KUKA KRL program: f1_Kuka_APT228T02S28.SRC

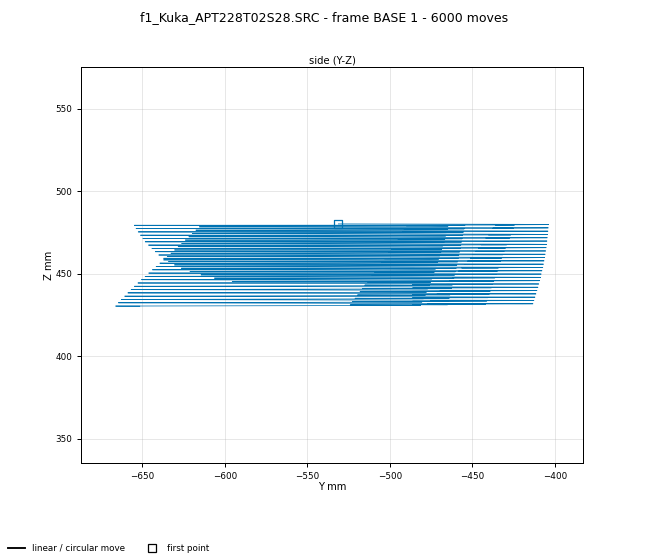
[picture p0: tool path of f1_Kuka_APT228T02S28.SRC in frame BASE 1, 6000 of 6001 moves have a stored position in this frame; points joined in program order, loops and branches not executed]
&ACCESS RVP
&REL 2
&PARAM TEMPLATE = C:\KRC\Roboter\Template\vorgabe
&PARAM EDITMASK = *
DEF f1_Kuka_APT228T02S28()


;FOLD INI;%{PE}%V3.2.0,%MKUKATPBASIS,%CINIT,%VCOMMON,%P
  ;FOLD BAS INI;%{E}%V3.2.0,%MKUKATPBASIS,%CINIT,%VINIT,%P
    GLOBAL INTERRUPT DECL 3 WHEN $STOPMESS==TRUE DO IR_STOPM ( )
    INTERRUPT ON 3
    BAS (#INITMOV,0 )
  ;ENDFOLD (BAS INI)
  ;FOLD USER INI;%{E}%V3.2.0,%MKUKATPUSER,%CINIT,%VINIT,%P
    ;Make your modifications here
  ;ENDFOLD (USER INI)
;ENDFOLD (INI)


;*** Make Null PTP Move
  PTP $pos_act

;*** Auto Load The Correct TOOL Data
  $tool=tool_data[2]

;*** Auto Load The Correct BASE Data
  $base=base_data[1]

  $ADVANCE = 5

;*** Restate Last Velocity
MMPM(30000.0)
SetRPM(8000)
LIN {X 0.012,Y -531.223,Z 480.140,A 0.000,B 0.000,C 90.000,E1 241.129} C_DIS
LIN {X -0.132,Y -524.473,Z 480.128,A 0.000,B 0.000,C 90.000,E1 239.125} C_DIS
LIN {X -0.042,Y -519.669,Z 480.120,A 0.000,B 0.000,C 90.000,E1 237.661} C_DIS
LIN {X -0.136,Y -515.820,Z 480.114,A 0.000,B 0.000,C 90.000,E1 236.501} C_DIS
LIN {X 0.003,Y -511.801,Z 480.107,A 0.000,B 0.000,C 90.000,E1 235.308} C_DIS
LIN {X 0.099,Y -503.620,Z 480.094,A 0.000,B 0.000,C 90.000,E1 232.924} C_DIS
LIN {X 0.015,Y -495.240,Z 480.079,A 0.000,B 0.000,C 90.000,E1 230.231} C_DIS
LIN {X 0.077,Y -489.925,Z 480.069,A 0.000,B 0.000,C 90.000,E1 228.405} C_DIS
LIN {X -0.155,Y -485.610,Z 480.061,A 0.000,B 0.000,C 90.000,E1 226.905} C_DIS
LIN {X 0.222,Y -481.353,Z 480.052,A 0.000,B 0.000,C 90.000,E1 225.324} C_DIS
LIN {X 0.174,Y -474.838,Z 480.038,A 0.000,B 0.000,C 90.000,E1 222.852} C_DIS
LIN {X -0.124,Y -469.500,Z 480.026,A 0.000,B 0.000,C 90.000,E1 220.701} C_DIS
LIN {X -0.093,Y -463.775,Z 480.012,A 0.000,B 0.000,C 90.000,E1 218.177} C_DIS
LIN {X 0.094,Y -459.135,Z 480.000,A 0.000,B 0.000,C 90.000,E1 215.931} C_DIS
LIN {X -0.017,Y -454.671,Z 479.987,A 0.000,B 0.000,C 90.000,E1 213.706} C_DIS
LIN {X -0.201,Y -450.942,Z 479.977,A 0.000,B 0.000,C 90.000,E1 211.799} C_DIS
LIN {X 0.216,Y -447.979,Z 479.968,A 0.000,B 0.000,C 90.000,E1 210.129} C_DIS
LIN {X -0.195,Y -444.403,Z 479.957,A 0.000,B 0.000,C 90.000,E1 208.231} C_DIS
LIN {X 0.099,Y -440.825,Z 479.946,A 0.000,B 0.000,C 90.000,E1 206.232} C_DIS
LIN {X 0.104,Y -437.235,Z 479.935,A 0.000,B 0.000,C 90.000,E1 204.259} C_DIS
LIN {X 0.071,Y -433.639,Z 479.924,A 0.000,B 0.000,C 90.000,E1 202.280} C_DIS
LIN {X -0.019,Y -428.986,Z 479.909,A 0.000,B 0.000,C 90.000,E1 199.631} C_DIS
LIN {X 0.061,Y -425.308,Z 479.896,A 0.000,B 0.000,C 90.000,E1 197.275} C_DIS
LIN {X 0.036,Y -421.007,Z 479.879,A 0.000,B 0.000,C 90.000,E1 194.245} C_DIS
LIN {X -0.197,Y -418.417,Z 479.868,A 0.000,B 0.000,C 90.000,E1 192.243} C_DIS
LIN {X -0.066,Y -415.176,Z 479.853,A 0.000,B 0.000,C 90.000,E1 189.500} C_DIS
LIN {X -0.177,Y -412.255,Z 479.838,A 0.000,B 0.000,C 90.000,E1 186.777} C_DIS
LIN {X -0.098,Y -409.929,Z 479.824,A 0.000,B 0.000,C 90.000,E1 184.359} C_DIS
LIN {X -0.138,Y -407.863,Z 479.811,A 0.000,B 0.000,C 90.000,E1 181.949} C_DIS
LIN {X 0.112,Y -405.824,Z 479.793,A 0.000,B 0.000,C 90.000,E1 178.797} C_DIS
LIN {X -0.117,Y -404.326,Z 479.774,A 0.000,B 0.000,C 90.000,E1 175.355} C_DIS
LIN {X 0.145,Y -403.885,Z 479.755,A 0.000,B 0.000,C 90.000,E1 171.837} C_DIS
LIN {X -0.149,Y -404.385,Z 479.735,A 0.000,B 0.000,C 90.000,E1 168.398} C_DIS
LIN {X 0.042,Y -405.380,Z 479.720,A 0.000,B 0.000,C 90.000,E1 165.589} C_DIS
LIN {X -0.122,Y -407.093,Z 479.703,A 0.000,B 0.000,C 90.000,E1 162.489} C_DIS
LIN {X -0.085,Y -408.847,Z 479.689,A 0.000,B 0.000,C 90.000,E1 160.061} C_DIS
LIN {X 0.144,Y -410.958,Z 479.676,A 0.000,B 0.000,C 90.000,E1 157.614} C_DIS
LIN {X 0.241,Y -413.011,Z 479.664,A 0.000,B 0.000,C 90.000,E1 155.537} C_DIS
LIN {X 0.018,Y -415.202,Z 479.653,A 0.000,B 0.000,C 90.000,E1 153.512} C_DIS
LIN {X -0.097,Y -417.093,Z 479.643,A 0.000,B 0.000,C 90.000,E1 151.820} C_DIS
LIN {X 0.146,Y -419.334,Z 479.632,A 0.000,B 0.000,C 90.000,E1 149.744} C_DIS
LIN {X -0.085,Y -421.583,Z 479.621,A 0.000,B 0.000,C 90.000,E1 147.740} C_DIS
LIN {X 0.013,Y -423.053,Z 479.613,A 0.000,B 0.000,C 90.000,E1 146.373} C_DIS
LIN {X 0.000,Y -424.931,Z 479.604,A 0.000,B 0.000,C 90.000,E1 144.689} C_DIS
LIN {X -0.113,Y -427.584,Z 479.591,A 0.000,B 0.000,C 90.000,E1 142.351} C_DIS
LIN {X 0.145,Y -429.546,Z 479.582,A 0.000,B 0.000,C 90.000,E1 140.642} C_DIS
LIN {X 0.089,Y -431.818,Z 479.570,A 0.000,B 0.000,C 90.000,E1 138.647} C_DIS
LIN {X 0.135,Y -433.268,Z 479.563,A 0.000,B 0.000,C 90.000,E1 137.310} C_DIS
LIN {X 0.207,Y -434.411,Z 479.556,A 0.000,B 0.000,C 90.000,E1 135.972} C_DIS
LIN {X 0.040,Y -435.117,Z 479.550,A 0.000,B 0.000,C 90.000,E1 135.000} C_DIS
LIN {X -0.120,Y -435.679,Z 479.545,A 0.000,B 0.000,C 90.000,E1 134.028} C_DIS
LIN {X 0.040,Y -436.073,Z 479.539,A 0.000,B 0.000,C 90.000,E1 133.014} C_DIS
LIN {X 0.208,Y -436.280,Z 479.534,A 0.000,B 0.000,C 90.000,E1 132.000} C_DIS
LIN {X -0.241,Y -436.121,Z 479.528,A 0.000,B 0.000,C 90.000,E1 131.067} C_DIS
LIN {X 0.250,Y -435.587,Z 479.523,A 0.000,B 0.000,C 90.000,E1 130.011} C_DIS
LIN {X -0.224,Y -434.407,Z 479.515,A 0.000,B 0.000,C 90.000,E1 128.749} C_DIS
LIN {X 0.045,Y -433.713,Z 479.511,A 0.000,B 0.000,C 90.000,E1 128.051} C_DIS
LIN {X 0.146,Y -431.523,Z 479.502,A 0.000,B 0.000,C 90.000,E1 126.377} C_DIS
LIN {X 0.291,Y -429.397,Z 479.495,A 0.000,B 0.000,C 90.000,E1 125.025} C_DIS
LIN {X 0.154,Y -427.076,Z 479.487,A 0.000,B 0.000,C 90.000,E1 123.706} C_DIS
LIN {X 0.257,Y -424.569,Z 479.480,A 0.000,B 0.000,C 90.000,E1 122.339} C_DIS
LIN {X 0.218,Y -424.582,Z 479.480,A 0.000,B 0.000,C 90.000,E1 122.339} C_DIS
LIN {X -0.108,Y -430.513,Z 479.469,A 0.000,B 0.000,C 90.000,E1 120.384} C_DIS
LIN {X 0.073,Y -433.632,Z 479.461,A 0.000,B 0.000,C 90.000,E1 119.027} C_DIS
LIN {X -0.054,Y -443.352,Z 479.441,A 0.000,B 0.000,C 90.000,E1 115.412} C_DIS
LIN {X -0.016,Y -444.339,Z 479.439,A 0.000,B 0.000,C 90.000,E1 115.079} C_DIS
LIN {X -0.162,Y -445.170,Z 479.438,A 0.000,B 0.000,C 90.000,E1 114.771} C_DIS
LIN {X -0.055,Y -454.357,Z 479.416,A 0.000,B 0.000,C 90.000,E1 110.865} C_DIS
LIN {X 0.066,Y -457.027,Z 479.411,A 0.000,B 0.000,C 90.000,E1 109.885} C_DIS
LIN {X 0.214,Y -458.867,Z 479.405,A 0.000,B 0.000,C 90.000,E1 108.906} C_DIS
LIN {X -0.129,Y -467.225,Z 479.384,A 0.000,B 0.000,C 90.000,E1 105.134} C_DIS
LIN {X 0.247,Y -467.938,Z 479.382,A 0.000,B 0.000,C 90.000,E1 104.773} C_DIS
LIN {X 0.127,Y -471.660,Z 479.369,A 0.000,B 0.000,C 90.000,E1 102.411} C_DIS
LIN {X 0.102,Y -487.037,Z 479.369,A 0.000,B 0.000,C 90.000,E1 102.411} C_DIS
LIN {X 0.072,Y -492.252,Z 479.369,A 0.000,B 0.000,C 90.000,E1 102.411} C_DIS
LIN {X -0.017,Y -505.550,Z 479.369,A 0.000,B 0.000,C 90.000,E1 102.355} C_DIS
LIN {X 0.021,Y -514.960,Z 479.368,A 0.000,B 0.000,C 90.000,E1 102.243} C_DIS
LIN {X 0.067,Y -529.400,Z 479.367,A 0.000,B 0.000,C 90.000,E1 102.007} C_DIS
LIN {X -0.010,Y -536.162,Z 479.366,A 0.000,B 0.000,C 90.000,E1 101.883} C_DIS
LIN {X -0.170,Y -546.119,Z 479.365,A 0.000,B 0.000,C 90.000,E1 101.658} C_DIS
LIN {X -0.263,Y -552.707,Z 479.364,A 0.000,B 0.000,C 90.000,E1 101.478} C_DIS
LIN {X -0.070,Y -559.550,Z 479.362,A 0.000,B 0.000,C 90.000,E1 101.243} C_DIS
LIN {X -0.128,Y -566.051,Z 479.361,A 0.000,B 0.000,C 90.000,E1 101.007} C_DIS
LIN {X -0.189,Y -575.852,Z 479.359,A 0.000,B 0.000,C 90.000,E1 100.602} C_DIS
LIN {X -0.232,Y -582.322,Z 479.357,A 0.000,B 0.000,C 90.000,E1 100.310} C_DIS
LIN {X -0.252,Y -590.194,Z 479.355,A 0.000,B 0.000,C 90.000,E1 99.905} C_DIS
LIN {X -0.314,Y -596.274,Z 479.353,A 0.000,B 0.000,C 90.000,E1 99.557} C_DIS
LIN {X -0.089,Y -602.333,Z 479.351,A 0.000,B 0.000,C 90.000,E1 99.151} C_DIS
LIN {X -0.119,Y -607.977,Z 479.349,A 0.000,B 0.000,C 90.000,E1 98.746} C_DIS
LIN {X 0.031,Y -610.636,Z 479.347,A 0.000,B 0.000,C 90.000,E1 98.511} C_DIS
LIN {X 0.024,Y -611.829,Z 479.347,A 0.000,B 0.000,C 90.000,E1 98.398} C_DIS
LIN {X 0.055,Y -614.172,Z 479.346,A 0.000,B 0.000,C 90.000,E1 98.219} C_DIS
LIN {X 0.072,Y -619.045,Z 479.343,A 0.000,B 0.000,C 90.000,E1 97.757} C_DIS
LIN {X 0.274,Y -625.534,Z 479.339,A 0.000,B 0.000,C 90.000,E1 97.068} C_DIS
LIN {X 0.306,Y -632.569,Z 479.335,A 0.000,B 0.000,C 90.000,E1 96.201} C_DIS
LIN {X -0.316,Y -636.839,Z 479.331,A 0.000,B 0.000,C 90.000,E1 95.625} C_DIS
LIN {X 0.242,Y -641.330,Z 479.327,A 0.000,B 0.000,C 90.000,E1 94.821} C_DIS
LIN {X -0.195,Y -643.986,Z 479.324,A 0.000,B 0.000,C 90.000,E1 94.359} C_DIS
LIN {X -0.210,Y -647.461,Z 479.320,A 0.000,B 0.000,C 90.000,E1 93.612} C_DIS
LIN {X 0.024,Y -649.407,Z 479.317,A 0.000,B 0.000,C 90.000,E1 93.094} C_DIS
LIN {X 0.238,Y -650.991,Z 479.314,A 0.000,B 0.000,C 90.000,E1 92.579} C_DIS
LIN {X 0.026,Y -651.725,Z 479.313,A 0.000,B 0.000,C 90.000,E1 92.350} C_DIS
LIN {X 0.263,Y -652.909,Z 479.310,A 0.000,B 0.000,C 90.000,E1 91.835} C_DIS
LIN {X -0.126,Y -653.794,Z 479.308,A 0.000,B 0.000,C 90.000,E1 91.375} C_DIS
LIN {X 0.126,Y -654.404,Z 479.305,A 0.000,B 0.000,C 90.000,E1 90.859} C_DIS
LIN {X -0.073,Y -654.659,Z 479.304,A 0.000,B 0.000,C 90.000,E1 90.630} C_DIS
LIN {X 0.187,Y -654.824,Z 479.301,A 0.000,B 0.000,C 90.000,E1 90.115} C_DIS
LIN {X 0.252,Y -654.511,Z 479.297,A 0.000,B 0.000,C 90.000,E1 89.370} C_DIS
LIN {X -0.142,Y -654.071,Z 479.294,A 0.000,B 0.000,C 90.000,E1 88.912} C_DIS
LIN {X 0.112,Y -653.331,Z 479.291,A 0.000,B 0.000,C 90.000,E1 88.396} C_DIS
LIN {X -0.269,Y -652.308,Z 479.288,A 0.000,B 0.000,C 90.000,E1 87.936} C_DIS
LIN {X -0.026,Y -650.976,Z 479.286,A 0.000,B 0.000,C 90.000,E1 87.421} C_DIS
LIN {X 0.203,Y -649.293,Z 479.283,A 0.000,B 0.000,C 90.000,E1 86.906} C_DIS
LIN {X -0.190,Y -647.401,Z 479.280,A 0.000,B 0.000,C 90.000,E1 86.445} C_DIS
LIN {X -0.172,Y -643.974,Z 479.276,A 0.000,B 0.000,C 90.000,E1 85.698} C_DIS
LIN {X -0.191,Y -639.704,Z 479.272,A 0.000,B 0.000,C 90.000,E1 84.951} C_DIS
LIN {X 0.003,Y -636.694,Z 479.269,A 0.000,B 0.000,C 90.000,E1 84.432} C_DIS
LIN {X -0.027,Y -631.495,Z 479.265,A 0.000,B 0.000,C 90.000,E1 83.685} C_DIS
LIN {X -0.108,Y -625.374,Z 479.261,A 0.000,B 0.000,C 90.000,E1 82.932} C_DIS
LIN {X -0.170,Y -619.575,Z 479.257,A 0.000,B 0.000,C 90.000,E1 82.299} C_DIS
LIN {X -0.080,Y -613.392,Z 479.254,A 0.000,B 0.000,C 90.000,E1 81.659} C_DIS
LIN {X 0.197,Y -608.136,Z 479.251,A 0.000,B 0.000,C 90.000,E1 81.141} C_DIS
LIN {X 0.113,Y -598.328,Z 479.246,A 0.000,B 0.000,C 90.000,E1 80.330} C_DIS
LIN {X 0.198,Y -596.955,Z 479.246,A 0.000,B 0.000,C 90.000,E1 80.208} C_DIS
LIN {X 0.131,Y -593.705,Z 479.244,A 0.000,B 0.000,C 90.000,E1 79.982} C_DIS
LIN {X 0.106,Y -591.339,Z 479.243,A 0.000,B 0.000,C 90.000,E1 79.803} C_DIS
LIN {X -0.030,Y -584.889,Z 479.241,A 0.000,B 0.000,C 90.000,E1 79.398} C_DIS
LIN {X 0.169,Y -578.243,Z 479.239,A 0.000,B 0.000,C 90.000,E1 78.993} C_DIS
LIN {X -0.120,Y -573.153,Z 479.238,A 0.000,B 0.000,C 90.000,E1 78.757} C_DIS
LIN {X 0.009,Y -567.505,Z 479.236,A 0.000,B 0.000,C 90.000,E1 78.522} C_DIS
LIN {X -0.060,Y -561.346,Z 479.235,A 0.000,B 0.000,C 90.000,E1 78.342} C_DIS
LIN {X -0.261,Y -555.145,Z 479.234,A 0.000,B 0.000,C 90.000,E1 78.229} C_DIS
LIN {X -0.189,Y -548.703,Z 479.234,A 0.000,B 0.000,C 90.000,E1 78.117} C_DIS
LIN {X -0.030,Y -542.488,Z 479.234,A 0.000,B 0.000,C 90.000,E1 78.049} C_DIS
LIN {X -0.116,Y -540.273,Z 479.234,A 0.000,B 0.000,C 90.000,E1 78.049} C_DIS
LIN {X -0.142,Y -481.260,Z 479.234,A 0.000,B 0.000,C 90.000,E1 78.049} C_DIS
LIN {X -0.168,Y -480.601,Z 479.228,A 0.000,B 0.000,C 90.000,E1 76.992} C_DIS
LIN {X 0.157,Y -480.228,Z 479.226,A 0.000,B 0.000,C 90.000,E1 76.645} C_DIS
LIN {X 0.046,Y -474.058,Z 479.200,A 0.000,B 0.000,C 90.000,E1 72.000} C_DIS
LIN {X 0.075,Y -465.491,Z 479.172,A 0.000,B 0.000,C 90.000,E1 66.975} C_DIS
LIN {X -0.145,Y -457.048,Z 479.149,A 0.000,B 0.000,C 90.000,E1 62.871} C_DIS
LIN {X -0.036,Y -455.462,Z 479.144,A 0.000,B 0.000,C 90.000,E1 61.897} C_DIS
LIN {X 0.070,Y -454.547,Z 479.142,A 0.000,B 0.000,C 90.000,E1 61.513} C_DIS
LIN {X 0.030,Y -454.555,Z 479.142,A 0.000,B 0.000,C 90.000,E1 61.513} C_DIS
LIN {X 0.119,Y -460.681,Z 479.136,A 0.000,B 0.000,C 90.000,E1 60.461} C_DIS
LIN {X 0.123,Y -465.104,Z 479.132,A 0.000,B 0.000,C 90.000,E1 59.665} C_DIS
LIN {X 0.173,Y -469.336,Z 479.127,A 0.000,B 0.000,C 90.000,E1 58.869} C_DIS
LIN {X 0.091,Y -471.678,Z 479.125,A 0.000,B 0.000,C 90.000,E1 58.408} C_DIS
LIN {X 0.021,Y -473.962,Z 479.122,A 0.000,B 0.000,C 90.000,E1 57.946} C_DIS
LIN {X 0.001,Y -477.214,Z 479.118,A 0.000,B 0.000,C 90.000,E1 57.168} C_DIS
LIN {X -0.012,Y -479.534,Z 479.114,A 0.000,B 0.000,C 90.000,E1 56.548} C_DIS
LIN {X -0.010,Y -481.447,Z 479.111,A 0.000,B 0.000,C 90.000,E1 55.928} C_DIS
LIN {X 0.006,Y -483.056,Z 479.107,A 0.000,B 0.000,C 90.000,E1 55.308} C_DIS
LIN {X 0.218,Y -483.824,Z 479.106,A 0.000,B 0.000,C 90.000,E1 54.975} C_DIS
LIN {X 0.071,Y -485.607,Z 479.100,A 0.000,B 0.000,C 90.000,E1 54.069} C_DIS
LIN {X 0.010,Y -486.605,Z 479.097,A 0.000,B 0.000,C 90.000,E1 53.463} C_DIS
LIN {X -0.108,Y -487.729,Z 479.092,A 0.000,B 0.000,C 90.000,E1 52.557} C_DIS
LIN {X 0.078,Y -488.561,Z 479.087,A 0.000,B 0.000,C 90.000,E1 51.618} C_DIS
LIN {X -0.272,Y -489.301,Z 479.080,A 0.000,B 0.000,C 90.000,E1 50.436} C_DIS
LIN {X 0.088,Y -489.649,Z 479.077,A 0.000,B 0.000,C 90.000,E1 49.784} C_DIS
LIN {X 0.065,Y -489.970,Z 479.070,A 0.000,B 0.000,C 90.000,E1 48.566} C_DIS
LIN {X 0.216,Y -490.114,Z 479.065,A 0.000,B 0.000,C 90.000,E1 47.634} C_DIS
LIN {X 0.012,Y -490.127,Z 479.060,A 0.000,B 0.000,C 90.000,E1 46.743} C_DIS
LIN {X -0.013,Y -489.993,Z 479.053,A 0.000,B 0.000,C 90.000,E1 45.526} C_DIS
LIN {X -0.074,Y -489.460,Z 479.043,A 0.000,B 0.000,C 90.000,E1 43.704} C_DIS
LIN {X 0.060,Y -488.649,Z 479.034,A 0.000,B 0.000,C 90.000,E1 42.162} C_DIS
LIN {X 0.178,Y -487.751,Z 479.026,A 0.000,B 0.000,C 90.000,E1 40.620} C_DIS
LIN {X -0.045,Y -486.642,Z 479.017,A 0.000,B 0.000,C 90.000,E1 39.116} C_DIS
LIN {X -0.091,Y -485.355,Z 479.007,A 0.000,B 0.000,C 90.000,E1 37.282} C_DIS
LIN {X 0.100,Y -484.171,Z 478.999,A 0.000,B 0.000,C 90.000,E1 35.724} C_DIS
LIN {X 0.175,Y -483.071,Z 478.992,A 0.000,B 0.000,C 90.000,E1 34.485} C_DIS
LIN {X -0.163,Y -481.831,Z 478.985,A 0.000,B 0.000,C 90.000,E1 33.293} C_DIS
LIN {X 0.041,Y -479.913,Z 478.975,A 0.000,B 0.000,C 90.000,E1 31.416} C_DIS
LIN {X 0.201,Y -477.833,Z 478.964,A 0.000,B 0.000,C 90.000,E1 29.539} C_DIS
LIN {X -0.010,Y -475.057,Z 478.950,A 0.000,B 0.000,C 90.000,E1 27.078} C_DIS
LIN {X -0.051,Y -472.807,Z 478.938,A 0.000,B 0.000,C 90.000,E1 24.899} C_DIS
LIN {X -0.021,Y -470.504,Z 478.923,A 0.000,B 0.000,C 90.000,E1 22.078} C_DIS
LIN {X -0.060,Y -469.133,Z 478.910,A 0.000,B 0.000,C 90.000,E1 19.885} C_DIS
LIN {X -0.135,Y -467.809,Z 478.898,A 0.000,B 0.000,C 90.000,E1 17.692} C_DIS
LIN {X -0.209,Y -467.149,Z 478.891,A 0.000,B 0.000,C 90.000,E1 16.441} C_DIS
LIN {X 0.148,Y -466.080,Z 478.879,A 0.000,B 0.000,C 90.000,E1 14.189} C_DIS
LIN {X 0.173,Y -465.202,Z 478.865,A 0.000,B 0.000,C 90.000,E1 11.658} C_DIS
LIN {X -0.082,Y -464.836,Z 478.854,A 0.000,B 0.000,C 90.000,E1 9.792} C_DIS
LIN {X -0.109,Y -464.762,Z 478.839,A 0.000,B 0.000,C 90.000,E1 6.947} C_DIS
LIN {X 0.108,Y -465.381,Z 478.823,A 0.000,B 0.000,C 90.000,E1 4.073} C_DIS
LIN {X -0.139,Y -466.810,Z 478.807,A 0.000,B 0.000,C 90.000,E1 1.260} C_DIS
LIN {X -0.051,Y -469.239,Z 478.790,A 0.000,B 0.000,C 90.000,E1 358.224} C_DIS
LIN {X 0.069,Y -471.793,Z 478.776,A 0.000,B 0.000,C 90.000,E1 355.698} C_DIS
LIN {X 0.021,Y -474.479,Z 478.764,A 0.000,B 0.000,C 90.000,E1 353.514} C_DIS
LIN {X 0.142,Y -477.400,Z 478.752,A 0.000,B 0.000,C 90.000,E1 351.319} C_DIS
LIN {X 0.211,Y -481.644,Z 478.736,A 0.000,B 0.000,C 90.000,E1 348.522} C_DIS
LIN {X -0.080,Y -488.580,Z 478.716,A 0.000,B 0.000,C 90.000,E1 344.866} C_DIS
LIN {X -0.028,Y -493.214,Z 478.704,A 0.000,B 0.000,C 90.000,E1 342.725} C_DIS
LIN {X -0.031,Y -498.081,Z 478.692,A 0.000,B 0.000,C 90.000,E1 340.604} C_DIS
LIN {X 0.268,Y -503.058,Z 478.681,A 0.000,B 0.000,C 90.000,E1 338.465} C_DIS
LIN {X 0.029,Y -506.563,Z 478.672,A 0.000,B 0.000,C 90.000,E1 336.997} C_DIS
LIN {X -0.217,Y -509.969,Z 478.664,A 0.000,B 0.000,C 90.000,E1 335.537} C_DIS
LIN {X 0.061,Y -514.686,Z 478.652,A 0.000,B 0.000,C 90.000,E1 333.435} C_DIS
LIN {X -0.004,Y -519.367,Z 478.641,A 0.000,B 0.000,C 90.000,E1 331.385} C_DIS
LIN {X 0.146,Y -523.507,Z 478.631,A 0.000,B 0.000,C 90.000,E1 329.616} C_DIS
LIN {X 0.167,Y -528.460,Z 478.620,A 0.000,B 0.000,C 90.000,E1 327.582} C_DIS
LIN {X -0.113,Y -532.759,Z 478.610,A 0.000,B 0.000,C 90.000,E1 325.881} C_DIS
LIN {X -0.013,Y -537.107,Z 478.601,A 0.000,B 0.000,C 90.000,E1 324.149} C_DIS
LIN {X 0.057,Y -541.507,Z 478.591,A 0.000,B 0.000,C 90.000,E1 322.431} C_DIS
LIN {X 0.069,Y -544.437,Z 478.585,A 0.000,B 0.000,C 90.000,E1 321.295} C_DIS
LIN {X -0.130,Y -548.833,Z 478.576,A 0.000,B 0.000,C 90.000,E1 319.622} C_DIS
LIN {X -0.366,Y -552.364,Z 478.568,A 0.000,B 0.000,C 90.000,E1 318.243} C_DIS
LIN {X -0.105,Y -556.598,Z 478.559,A 0.000,B 0.000,C 90.000,E1 316.539} C_DIS
LIN {X -0.344,Y -558.647,Z 478.554,A 0.000,B 0.000,C 90.000,E1 315.729} C_DIS
LIN {X -0.289,Y -563.373,Z 478.543,A 0.000,B 0.000,C 90.000,E1 313.785} C_DIS
LIN {X 0.115,Y -566.743,Z 478.535,A 0.000,B 0.000,C 90.000,E1 312.366} C_DIS
LIN {X 0.198,Y -570.113,Z 478.528,A 0.000,B 0.000,C 90.000,E1 310.987} C_DIS
LIN {X 0.105,Y -574.054,Z 478.519,A 0.000,B 0.000,C 90.000,E1 309.358} C_DIS
LIN {X -0.058,Y -577.354,Z 478.511,A 0.000,B 0.000,C 90.000,E1 308.016} C_DIS
LIN {X -0.067,Y -580.696,Z 478.504,A 0.000,B 0.000,C 90.000,E1 306.664} C_DIS
LIN {X 0.167,Y -584.645,Z 478.495,A 0.000,B 0.000,C 90.000,E1 305.025} C_DIS
LIN {X -0.053,Y -587.924,Z 478.487,A 0.000,B 0.000,C 90.000,E1 303.706} C_DIS
LIN {X 0.274,Y -591.153,Z 478.480,A 0.000,B 0.000,C 90.000,E1 302.339} C_DIS
LIN {X -0.364,Y -593.589,Z 478.474,A 0.000,B 0.000,C 90.000,E1 301.337} C_DIS
LIN {X -0.157,Y -595.818,Z 478.468,A 0.000,B 0.000,C 90.000,E1 300.256} C_DIS
LIN {X -0.222,Y -597.922,Z 478.462,A 0.000,B 0.000,C 90.000,E1 299.205} C_DIS
LIN {X 0.194,Y -600.396,Z 478.455,A 0.000,B 0.000,C 90.000,E1 297.847} C_DIS
LIN {X -0.086,Y -602.210,Z 478.449,A 0.000,B 0.000,C 90.000,E1 296.821} C_DIS
LIN {X -0.077,Y -603.809,Z 478.443,A 0.000,B 0.000,C 90.000,E1 295.771} C_DIS
LIN {X -0.030,Y -605.166,Z 478.437,A 0.000,B 0.000,C 90.000,E1 294.719} C_DIS
LIN {X 0.297,Y -606.400,Z 478.432,A 0.000,B 0.000,C 90.000,E1 293.643} C_DIS
LIN {X 0.057,Y -608.086,Z 478.423,A 0.000,B 0.000,C 90.000,E1 292.099} C_DIS
LIN {X 0.182,Y -609.164,Z 478.417,A 0.000,B 0.000,C 90.000,E1 291.046} C_DIS
LIN {X 0.047,Y -610.357,Z 478.410,A 0.000,B 0.000,C 90.000,E1 289.758} C_DIS
LIN {X 0.243,Y -611.575,Z 478.401,A 0.000,B 0.000,C 90.000,E1 288.181} C_DIS
LIN {X -0.063,Y -612.618,Z 478.394,A 0.000,B 0.000,C 90.000,E1 286.913} C_DIS
LIN {X 0.055,Y -613.490,Z 478.387,A 0.000,B 0.000,C 90.000,E1 285.607} C_DIS
LIN {X 0.192,Y -614.173,Z 478.380,A 0.000,B 0.000,C 90.000,E1 284.300} C_DIS
LIN {X -0.169,Y -614.691,Z 478.374,A 0.000,B 0.000,C 90.000,E1 283.300} C_DIS
LIN {X 0.204,Y -615.238,Z 478.365,A 0.000,B 0.000,C 90.000,E1 281.715} C_DIS
LIN {X -0.152,Y -615.393,Z 478.359,A 0.000,B 0.000,C 90.000,E1 280.715} C_DIS
LIN {X 0.342,Y -615.445,Z 478.352,A 0.000,B 0.000,C 90.000,E1 279.378} C_DIS
LIN {X 0.135,Y -615.252,Z 478.345,A 0.000,B 0.000,C 90.000,E1 278.106} C_DIS
LIN {X -0.094,Y -615.018,Z 478.341,A 0.000,B 0.000,C 90.000,E1 277.352} C_DIS
LIN {X 0.233,Y -614.415,Z 478.334,A 0.000,B 0.000,C 90.000,E1 276.030} C_DIS
LIN {X -0.013,Y -613.883,Z 478.329,A 0.000,B 0.000,C 90.000,E1 275.277} C_DIS
LIN {X -0.038,Y -612.991,Z 478.324,A 0.000,B 0.000,C 90.000,E1 274.245} C_DIS
LIN {X 0.255,Y -612.193,Z 478.319,A 0.000,B 0.000,C 90.000,E1 273.440} C_DIS
LIN {X 0.212,Y -610.935,Z 478.314,A 0.000,B 0.000,C 90.000,E1 272.407} C_DIS
LIN {X 0.145,Y -609.502,Z 478.308,A 0.000,B 0.000,C 90.000,E1 271.375} C_DIS
LIN {X -0.014,Y -607.101,Z 478.299,A 0.000,B 0.000,C 90.000,E1 269.828} C_DIS
LIN {X 0.118,Y -604.861,Z 478.292,A 0.000,B 0.000,C 90.000,E1 268.511} C_DIS
LIN {X 0.223,Y -602.489,Z 478.285,A 0.000,B 0.000,C 90.000,E1 267.192} C_DIS
LIN {X 0.044,Y -600.479,Z 478.279,A 0.000,B 0.000,C 90.000,E1 266.159} C_DIS
LIN {X 0.113,Y -597.785,Z 478.271,A 0.000,B 0.000,C 90.000,E1 264.837} C_DIS
LIN {X -0.183,Y -594.350,Z 478.263,A 0.000,B 0.000,C 90.000,E1 263.280} C_DIS
LIN {X 0.117,Y -590.816,Z 478.254,A 0.000,B 0.000,C 90.000,E1 261.659} C_DIS
LIN {X 0.082,Y -587.844,Z 478.246,A 0.000,B 0.000,C 90.000,E1 260.330} C_DIS
LIN {X -0.246,Y -584.051,Z 478.237,A 0.000,B 0.000,C 90.000,E1 258.757} C_DIS
LIN {X 0.139,Y -581.394,Z 478.231,A 0.000,B 0.000,C 90.000,E1 257.645} C_DIS
LIN {X -0.068,Y -577.382,Z 478.223,A 0.000,B 0.000,C 90.000,E1 256.047} C_DIS
LIN {X 0.205,Y -573.198,Z 478.213,A 0.000,B 0.000,C 90.000,E1 254.393} C_DIS
LIN {X 0.013,Y -570.354,Z 478.207,A 0.000,B 0.000,C 90.000,E1 253.323} C_DIS
LIN {X 0.110,Y -566.649,Z 478.200,A 0.000,B 0.000,C 90.000,E1 251.945} C_DIS
LIN {X -0.010,Y -563.501,Z 478.194,A 0.000,B 0.000,C 90.000,E1 250.859} C_DIS
LIN {X 0.018,Y -560.269,Z 478.188,A 0.000,B 0.000,C 90.000,E1 249.752} C_DIS
LIN {X 0.101,Y -556.092,Z 478.180,A 0.000,B 0.000,C 90.000,E1 248.358} C_DIS
LIN {X 0.005,Y -551.678,Z 478.172,A 0.000,B 0.000,C 90.000,E1 246.975} C_DIS
LIN {X -0.140,Y -547.987,Z 478.166,A 0.000,B 0.000,C 90.000,E1 245.869} C_DIS
LIN {X -0.139,Y -543.199,Z 478.158,A 0.000,B 0.000,C 90.000,E1 244.460} C_DIS
LIN {X 0.000,Y -537.372,Z 478.149,A 0.000,B 0.000,C 90.000,E1 242.743} C_DIS
LIN {X 0.064,Y -532.582,Z 478.141,A 0.000,B 0.000,C 90.000,E1 241.307} C_DIS
LIN {X 0.147,Y -525.769,Z 478.129,A 0.000,B 0.000,C 90.000,E1 239.282} C_DIS
LIN {X -0.191,Y -520.940,Z 478.121,A 0.000,B 0.000,C 90.000,E1 237.867} C_DIS
LIN {X 0.100,Y -516.109,Z 478.113,A 0.000,B 0.000,C 90.000,E1 236.373} C_DIS
LIN {X 0.238,Y -512.066,Z 478.107,A 0.000,B 0.000,C 90.000,E1 235.182} C_DIS
LIN {X 0.131,Y -505.857,Z 478.097,A 0.000,B 0.000,C 90.000,E1 233.417} C_DIS
LIN {X -0.005,Y -496.365,Z 478.080,A 0.000,B 0.000,C 90.000,E1 230.436} C_DIS
LIN {X 0.089,Y -491.068,Z 478.070,A 0.000,B 0.000,C 90.000,E1 228.609} C_DIS
LIN {X 0.060,Y -485.853,Z 478.060,A 0.000,B 0.000,C 90.000,E1 226.782} C_DIS
LIN {X 0.222,Y -480.731,Z 478.050,A 0.000,B 0.000,C 90.000,E1 224.919} C_DIS
LIN {X -0.060,Y -475.869,Z 478.039,A 0.000,B 0.000,C 90.000,E1 223.095} C_DIS
LIN {X -0.242,Y -469.725,Z 478.026,A 0.000,B 0.000,C 90.000,E1 220.620} C_DIS
LIN {X 0.035,Y -464.728,Z 478.013,A 0.000,B 0.000,C 90.000,E1 218.382} C_DIS
LIN {X -0.016,Y -459.369,Z 477.999,A 0.000,B 0.000,C 90.000,E1 215.851} C_DIS
LIN {X -0.123,Y -454.908,Z 477.987,A 0.000,B 0.000,C 90.000,E1 213.627} C_DIS
LIN {X -0.131,Y -450.020,Z 477.972,A 0.000,B 0.000,C 90.000,E1 211.052} C_DIS
LIN {X 0.041,Y -446.990,Z 477.963,A 0.000,B 0.000,C 90.000,E1 209.411} C_DIS
LIN {X 0.005,Y -443.454,Z 477.953,A 0.000,B 0.000,C 90.000,E1 207.462} C_DIS
LIN {X -0.004,Y -441.028,Z 477.945,A 0.000,B 0.000,C 90.000,E1 206.155} C_DIS
LIN {X -0.179,Y -437.418,Z 477.934,A 0.000,B 0.000,C 90.000,E1 204.207} C_DIS
LIN {X -0.036,Y -433.794,Z 477.923,A 0.000,B 0.000,C 90.000,E1 202.206} C_DIS
LIN {X -0.063,Y -428.598,Z 477.907,A 0.000,B 0.000,C 90.000,E1 199.214} C_DIS
LIN {X 0.153,Y -425.965,Z 477.897,A 0.000,B 0.000,C 90.000,E1 197.511} C_DIS
LIN {X 0.145,Y -421.579,Z 477.881,A 0.000,B 0.000,C 90.000,E1 194.481} C_DIS
LIN {X -0.075,Y -418.963,Z 477.869,A 0.000,B 0.000,C 90.000,E1 192.479} C_DIS
LIN {X 0.147,Y -415.686,Z 477.854,A 0.000,B 0.000,C 90.000,E1 189.726} C_DIS
LIN {X 0.038,Y -412.707,Z 477.839,A 0.000,B 0.000,C 90.000,E1 187.004} C_DIS
LIN {X 0.097,Y -410.661,Z 477.828,A 0.000,B 0.000,C 90.000,E1 184.935} C_DIS
LIN {X 0.099,Y -408.517,Z 477.814,A 0.000,B 0.000,C 90.000,E1 182.522} C_DIS
LIN {X -0.037,Y -406.334,Z 477.797,A 0.000,B 0.000,C 90.000,E1 179.427} C_DIS
LIN {X 0.139,Y -404.706,Z 477.778,A 0.000,B 0.000,C 90.000,E1 175.931} C_DIS
LIN {X 0.008,Y -404.075,Z 477.762,A 0.000,B 0.000,C 90.000,E1 173.166} C_DIS
LIN {X -0.032,Y -404.074,Z 477.749,A 0.000,B 0.000,C 90.000,E1 170.735} C_DIS
LIN {X 0.069,Y -404.639,Z 477.733,A 0.000,B 0.000,C 90.000,E1 167.937} C_DIS
LIN {X -0.038,Y -405.813,Z 477.718,A 0.000,B 0.000,C 90.000,E1 165.172} C_DIS
LIN {X 0.053,Y -407.846,Z 477.698,A 0.000,B 0.000,C 90.000,E1 161.692} C_DIS
LIN {X -0.015,Y -410.380,Z 477.681,A 0.000,B 0.000,C 90.000,E1 158.592} C_DIS
LIN {X -0.055,Y -413.070,Z 477.666,A 0.000,B 0.000,C 90.000,E1 155.845} C_DIS
LIN {X 0.099,Y -415.277,Z 477.654,A 0.000,B 0.000,C 90.000,E1 153.768} C_DIS
LIN {X 0.105,Y -417.561,Z 477.643,A 0.000,B 0.000,C 90.000,E1 151.719} C_DIS
LIN {X 0.236,Y -419.506,Z 477.634,A 0.000,B 0.000,C 90.000,E1 149.999} C_DIS
LIN {X 0.016,Y -421.801,Z 477.622,A 0.000,B 0.000,C 90.000,E1 147.995} C_DIS
LIN {X 0.094,Y -423.693,Z 477.613,A 0.000,B 0.000,C 90.000,E1 146.294} C_DIS
LIN {X 0.072,Y -426.032,Z 477.602,A 0.000,B 0.000,C 90.000,E1 144.276} C_DIS
LIN {X 0.009,Y -428.408,Z 477.590,A 0.000,B 0.000,C 90.000,E1 142.271} C_DIS
LIN {X 0.015,Y -430.473,Z 477.581,A 0.000,B 0.000,C 90.000,E1 140.598} C_DIS
LIN {X 0.076,Y -432.061,Z 477.574,A 0.000,B 0.000,C 90.000,E1 139.256} C_DIS
LIN {X 0.124,Y -433.552,Z 477.566,A 0.000,B 0.000,C 90.000,E1 137.919} C_DIS
LIN {X -0.035,Y -434.715,Z 477.561,A 0.000,B 0.000,C 90.000,E1 136.944} C_DIS
LIN {X -0.257,Y -435.862,Z 477.553,A 0.000,B 0.000,C 90.000,E1 135.648} C_DIS
LIN {X 0.160,Y -436.771,Z 477.546,A 0.000,B 0.000,C 90.000,E1 134.271} C_DIS
LIN {X -0.032,Y -437.360,Z 477.539,A 0.000,B 0.000,C 90.000,E1 132.975} C_DIS
LIN {X -0.148,Y -437.647,Z 477.533,A 0.000,B 0.000,C 90.000,E1 132.000} C_DIS
LIN {X 0.035,Y -437.502,Z 477.528,A 0.000,B 0.000,C 90.000,E1 130.987} C_DIS
LIN {X -0.073,Y -436.962,Z 477.522,A 0.000,B 0.000,C 90.000,E1 130.011} C_DIS
LIN {X 0.088,Y -435.848,Z 477.515,A 0.000,B 0.000,C 90.000,E1 128.669} C_DIS
LIN {X 0.031,Y -434.702,Z 477.509,A 0.000,B 0.000,C 90.000,E1 127.684} C_DIS
LIN {X -0.118,Y -433.423,Z 477.504,A 0.000,B 0.000,C 90.000,E1 126.710} C_DIS
LIN {X -0.195,Y -431.332,Z 477.497,A 0.000,B 0.000,C 90.000,E1 125.391} C_DIS
LIN {X -0.055,Y -429.012,Z 477.489,A 0.000,B 0.000,C 90.000,E1 124.040} C_DIS
LIN {X 0.145,Y -425.849,Z 477.480,A 0.000,B 0.000,C 90.000,E1 122.339} C_DIS
LIN {X -0.191,Y -425.337,Z 477.478,A 0.000,B 0.000,C 90.000,E1 122.133} C_DIS
LIN {X 0.130,Y -425.335,Z 477.478,A 0.000,B 0.000,C 90.000,E1 122.084} C_DIS
LIN {X 0.079,Y -430.591,Z 477.469,A 0.000,B 0.000,C 90.000,E1 120.335} C_DIS
LIN {X 0.074,Y -441.499,Z 477.445,A 0.000,B 0.000,C 90.000,E1 116.027} C_DIS
LIN {X 0.200,Y -444.412,Z 477.439,A 0.000,B 0.000,C 90.000,E1 115.027} C_DIS
LIN {X 0.100,Y -445.896,Z 477.436,A 0.000,B 0.000,C 90.000,E1 114.387} C_DIS
LIN {X 0.237,Y -455.295,Z 477.414,A 0.000,B 0.000,C 90.000,E1 110.482} C_DIS
LIN {X -0.124,Y -457.095,Z 477.410,A 0.000,B 0.000,C 90.000,E1 109.885} C_DIS
LIN {X -0.119,Y -466.498,Z 477.386,A 0.000,B 0.000,C 90.000,E1 105.426} C_DIS
LIN {X 0.057,Y -467.970,Z 477.382,A 0.000,B 0.000,C 90.000,E1 104.773} C_DIS
LIN {X 0.167,Y -472.578,Z 477.366,A 0.000,B 0.000,C 90.000,E1 101.895} C_DIS
LIN {X 0.124,Y -495.393,Z 477.366,A 0.000,B 0.000,C 90.000,E1 101.895} C_DIS
LIN {X 0.086,Y -496.685,Z 477.366,A 0.000,B 0.000,C 90.000,E1 101.895} C_DIS
LIN {X 0.151,Y -501.518,Z 477.366,A 0.000,B 0.000,C 90.000,E1 101.883} C_DIS
LIN {X 0.073,Y -505.701,Z 477.366,A 0.000,B 0.000,C 90.000,E1 101.883} C_DIS
LIN {X 0.263,Y -517.560,Z 477.366,A 0.000,B 0.000,C 90.000,E1 101.771} C_DIS
LIN {X 0.083,Y -526.964,Z 477.365,A 0.000,B 0.000,C 90.000,E1 101.658} C_DIS
LIN {X -0.186,Y -529.308,Z 477.365,A 0.000,B 0.000,C 90.000,E1 101.658} C_DIS
LIN {X -0.137,Y -535.640,Z 477.364,A 0.000,B 0.000,C 90.000,E1 101.535} C_DIS
LIN {X -0.027,Y -545.715,Z 477.363,A 0.000,B 0.000,C 90.000,E1 101.299} C_DIS
LIN {X -0.115,Y -552.234,Z 477.362,A 0.000,B 0.000,C 90.000,E1 101.130} C_DIS
LIN {X 0.180,Y -559.121,Z 477.361,A 0.000,B 0.000,C 90.000,E1 100.894} C_DIS
LIN {X 0.282,Y -565.493,Z 477.359,A 0.000,B 0.000,C 90.000,E1 100.658} C_DIS
LIN {X 0.124,Y -568.993,Z 477.359,A 0.000,B 0.000,C 90.000,E1 100.546} C_DIS
LIN {X -0.164,Y -575.586,Z 477.357,A 0.000,B 0.000,C 90.000,E1 100.310} C_DIS
LIN {X -0.267,Y -583.593,Z 477.355,A 0.000,B 0.000,C 90.000,E1 99.962} C_DIS
LIN {X 0.036,Y -589.866,Z 477.353,A 0.000,B 0.000,C 90.000,E1 99.613} C_DIS
LIN {X -0.192,Y -594.663,Z 477.352,A 0.000,B 0.000,C 90.000,E1 99.378} C_DIS
LIN {X -0.148,Y -601.990,Z 477.350,A 0.000,B 0.000,C 90.000,E1 98.916} C_DIS
LIN {X -0.200,Y -606.470,Z 477.348,A 0.000,B 0.000,C 90.000,E1 98.624} C_DIS
LIN {X 0.175,Y -610.102,Z 477.346,A 0.000,B 0.000,C 90.000,E1 98.276} C_DIS
LIN {X 0.232,Y -613.295,Z 477.345,A 0.000,B 0.000,C 90.000,E1 98.049} C_DIS
LIN {X 0.259,Y -620.113,Z 477.341,A 0.000,B 0.000,C 90.000,E1 97.409} C_DIS
LIN {X 0.069,Y -625.859,Z 477.338,A 0.000,B 0.000,C 90.000,E1 96.834} C_DIS
LIN {X -0.021,Y -632.126,Z 477.334,A 0.000,B 0.000,C 90.000,E1 96.087} C_DIS
LIN {X -0.086,Y -637.249,Z 477.330,A 0.000,B 0.000,C 90.000,E1 95.334} C_DIS
LIN {X -0.039,Y -641.000,Z 477.326,A 0.000,B 0.000,C 90.000,E1 94.702} C_DIS
LIN {X -0.010,Y -644.236,Z 477.323,A 0.000,B 0.000,C 90.000,E1 94.073} C_DIS
LIN {X 0.210,Y -646.537,Z 477.320,A 0.000,B 0.000,C 90.000,E1 93.555} C_DIS
LIN {X -0.208,Y -648.482,Z 477.317,A 0.000,B 0.000,C 90.000,E1 93.094} C_DIS
LIN {X -0.001,Y -650.063,Z 477.314,A 0.000,B 0.000,C 90.000,E1 92.579} C_DIS
LIN {X 0.222,Y -651.379,Z 477.312,A 0.000,B 0.000,C 90.000,E1 92.064} C_DIS
LIN {X 0.013,Y -651.989,Z 477.310,A 0.000,B 0.000,C 90.000,E1 91.835} C_DIS
LIN {X 0.271,Y -652.834,Z 477.307,A 0.000,B 0.000,C 90.000,E1 91.318} C_DIS
LIN {X 0.316,Y -653.664,Z 477.303,A 0.000,B 0.000,C 90.000,E1 90.573} C_DIS
LIN {X -0.085,Y -653.805,Z 477.301,A 0.000,B 0.000,C 90.000,E1 90.115} C_DIS
LIN {X -0.030,Y -653.420,Z 477.297,A 0.000,B 0.000,C 90.000,E1 89.370} C_DIS
LIN {X 0.222,Y -652.944,Z 477.294,A 0.000,B 0.000,C 90.000,E1 88.854} C_DIS
LIN {X -0.183,Y -652.106,Z 477.291,A 0.000,B 0.000,C 90.000,E1 88.396} C_DIS
LIN {X 0.079,Y -651.008,Z 477.288,A 0.000,B 0.000,C 90.000,E1 87.879} C_DIS
LIN {X -0.128,Y -650.362,Z 477.287,A 0.000,B 0.000,C 90.000,E1 87.650} C_DIS
LIN {X 0.099,Y -648.760,Z 477.284,A 0.000,B 0.000,C 90.000,E1 87.135} C_DIS
LIN {X -0.298,Y -646.844,Z 477.281,A 0.000,B 0.000,C 90.000,E1 86.674} C_DIS
LIN {X -0.099,Y -644.581,Z 477.279,A 0.000,B 0.000,C 90.000,E1 86.159} C_DIS
LIN {X 0.243,Y -642.750,Z 477.277,A 0.000,B 0.000,C 90.000,E1 85.755} C_DIS
LIN {X -0.044,Y -636.957,Z 477.271,A 0.000,B 0.000,C 90.000,E1 84.780} C_DIS
LIN {X -0.149,Y -630.747,Z 477.266,A 0.000,B 0.000,C 90.000,E1 83.913} C_DIS
LIN {X -0.309,Y -624.685,Z 477.262,A 0.000,B 0.000,C 90.000,E1 83.166} C_DIS
LIN {X 0.318,Y -618.802,Z 477.258,A 0.000,B 0.000,C 90.000,E1 82.470} C_DIS
LIN {X -0.241,Y -612.496,Z 477.255,A 0.000,B 0.000,C 90.000,E1 81.894} C_DIS
LIN {X 0.099,Y -607.210,Z 477.252,A 0.000,B 0.000,C 90.000,E1 81.376} C_DIS
LIN {X 0.073,Y -600.156,Z 477.249,A 0.000,B 0.000,C 90.000,E1 80.792} C_DIS
LIN {X 0.192,Y -595.811,Z 477.247,A 0.000,B 0.000,C 90.000,E1 80.443} C_DIS
LIN {X -0.085,Y -589.669,Z 477.245,A 0.000,B 0.000,C 90.000,E1 80.038} C_DIS
LIN {X -0.219,Y -584.774,Z 477.243,A 0.000,B 0.000,C 90.000,E1 79.746} C_DIS
LIN {X 0.144,Y -578.244,Z 477.241,A 0.000,B 0.000,C 90.000,E1 79.342} C_DIS
LIN {X -0.018,Y -573.004,Z 477.240,A 0.000,B 0.000,C 90.000,E1 79.106} C_DIS
LIN {X 0.241,Y -566.020,Z 477.238,A 0.000,B 0.000,C 90.000,E1 78.814} C_DIS
LIN {X 0.137,Y -558.974,Z 477.237,A 0.000,B 0.000,C 90.000,E1 78.634} C_DIS
LIN {X -0.129,Y -554.146,Z 477.237,A 0.000,B 0.000,C 90.000,E1 78.578} C_DIS
LIN {X 0.094,Y -547.205,Z 477.236,A 0.000,B 0.000,C 90.000,E1 78.465} C_DIS
LIN {X -0.120,Y -540.682,Z 477.236,A 0.000,B 0.000,C 90.000,E1 78.465} C_DIS
LIN {X -0.134,Y -481.566,Z 477.236,A 0.000,B 0.000,C 90.000,E1 78.465} C_DIS
LIN {X 0.128,Y -480.658,Z 477.228,A 0.000,B 0.000,C 90.000,E1 77.061} C_DIS
LIN {X 0.094,Y -480.404,Z 477.227,A 0.000,B 0.000,C 90.000,E1 76.756} C_DIS
LIN {X -0.133,Y -474.188,Z 477.201,A 0.000,B 0.000,C 90.000,E1 72.127} C_DIS
LIN {X 0.063,Y -472.384,Z 477.195,A 0.000,B 0.000,C 90.000,E1 71.167} C_DIS
LIN {X -0.100,Y -465.690,Z 477.173,A 0.000,B 0.000,C 90.000,E1 67.102} C_DIS
LIN {X 0.101,Y -456.156,Z 477.146,A 0.000,B 0.000,C 90.000,E1 62.308} C_DIS
LIN {X -0.071,Y -455.151,Z 477.143,A 0.000,B 0.000,C 90.000,E1 61.769} C_DIS
LIN {X 0.011,Y -455.048,Z 477.143,A 0.000,B 0.000,C 90.000,E1 61.719} C_DIS
LIN {X -0.029,Y -455.069,Z 477.143,A 0.000,B 0.000,C 90.000,E1 61.719} C_DIS
LIN {X 0.013,Y -461.067,Z 477.137,A 0.000,B 0.000,C 90.000,E1 60.717} C_DIS
LIN {X 0.024,Y -465.582,Z 477.133,A 0.000,B 0.000,C 90.000,E1 59.921} C_DIS
LIN {X 0.077,Y -469.869,Z 477.129,A 0.000,B 0.000,C 90.000,E1 59.125} C_DIS
LIN {X -0.240,Y -473.034,Z 477.125,A 0.000,B 0.000,C 90.000,E1 58.535} C_DIS
LIN {X -0.051,Y -475.361,Z 477.122,A 0.000,B 0.000,C 90.000,E1 58.043} C_DIS
LIN {X 0.092,Y -478.630,Z 477.118,A 0.000,B 0.000,C 90.000,E1 57.248} C_DIS
LIN {X 0.088,Y -480.968,Z 477.115,A 0.000,B 0.000,C 90.000,E1 56.628} C_DIS
LIN {X 0.100,Y -482.867,Z 477.111,A 0.000,B 0.000,C 90.000,E1 56.008} C_DIS
LIN {X -0.054,Y -485.244,Z 477.106,A 0.000,B 0.000,C 90.000,E1 55.102} C_DIS
LIN {X -0.183,Y -487.032,Z 477.101,A 0.000,B 0.000,C 90.000,E1 54.196} C_DIS
LIN {X 0.161,Y -488.048,Z 477.098,A 0.000,B 0.000,C 90.000,E1 53.543} C_DIS
LIN {X 0.058,Y -489.144,Z 477.093,A 0.000,B 0.000,C 90.000,E1 52.637} C_DIS
LIN {X -0.125,Y -489.946,Z 477.087,A 0.000,B 0.000,C 90.000,E1 51.743} C_DIS
LIN {X 0.087,Y -490.514,Z 477.082,A 0.000,B 0.000,C 90.000,E1 50.803} C_DIS
LIN {X 0.081,Y -491.022,Z 477.076,A 0.000,B 0.000,C 90.000,E1 49.585} C_DIS
LIN {X -0.075,Y -491.233,Z 477.070,A 0.000,B 0.000,C 90.000,E1 48.690} C_DIS
LIN {X 0.095,Y -491.332,Z 477.065,A 0.000,B 0.000,C 90.000,E1 47.757} C_DIS
LIN {X -0.070,Y -491.306,Z 477.060,A 0.000,B 0.000,C 90.000,E1 46.863} C_DIS
LIN {X -0.091,Y -491.113,Z 477.054,A 0.000,B 0.000,C 90.000,E1 45.648} C_DIS
LIN {X 0.057,Y -490.633,Z 477.045,A 0.000,B 0.000,C 90.000,E1 44.109} C_DIS
LIN {X -0.139,Y -490.237,Z 477.040,A 0.000,B 0.000,C 90.000,E1 43.218} C_DIS
LIN {X 0.005,Y -489.352,Z 477.032,A 0.000,B 0.000,C 90.000,E1 41.676} C_DIS
LIN {X -0.020,Y -488.558,Z 477.025,A 0.000,B 0.000,C 90.000,E1 40.458} C_DIS
LIN {X -0.019,Y -487.221,Z 477.015,A 0.000,B 0.000,C 90.000,E1 38.624} C_DIS
LIN {X 0.122,Y -486.091,Z 477.006,A 0.000,B 0.000,C 90.000,E1 37.076} C_DIS
LIN {X -0.173,Y -485.133,Z 476.999,A 0.000,B 0.000,C 90.000,E1 35.884} C_DIS
LIN {X 0.017,Y -483.731,Z 476.991,A 0.000,B 0.000,C 90.000,E1 34.326} C_DIS
LIN {X 0.112,Y -481.822,Z 476.980,A 0.000,B 0.000,C 90.000,E1 32.467} C_DIS
LIN {X 0.101,Y -480.145,Z 476.972,A 0.000,B 0.000,C 90.000,E1 30.924} C_DIS
LIN {X -0.181,Y -478.399,Z 476.963,A 0.000,B 0.000,C 90.000,E1 29.411} C_DIS
LIN {X -0.155,Y -475.600,Z 476.950,A 0.000,B 0.000,C 90.000,E1 26.924} C_DIS
LIN {X 0.033,Y -473.349,Z 476.937,A 0.000,B 0.000,C 90.000,E1 24.719} C_DIS
LIN {X 0.088,Y -471.067,Z 476.922,A 0.000,B 0.000,C 90.000,E1 21.897} C_DIS
LIN {X 0.066,Y -469.680,Z 476.910,A 0.000,B 0.000,C 90.000,E1 19.704} C_DIS
LIN {X 0.006,Y -468.369,Z 476.897,A 0.000,B 0.000,C 90.000,E1 17.511} C_DIS
LIN {X -0.061,Y -467.691,Z 476.890,A 0.000,B 0.000,C 90.000,E1 16.260} C_DIS
LIN {X 0.116,Y -466.471,Z 476.876,A 0.000,B 0.000,C 90.000,E1 13.716} C_DIS
LIN {X -0.046,Y -465.583,Z 476.861,A 0.000,B 0.000,C 90.000,E1 10.894} C_DIS
LIN {X 0.151,Y -465.194,Z 476.846,A 0.000,B 0.000,C 90.000,E1 8.341} C_DIS
LIN {X -0.191,Y -465.363,Z 476.832,A 0.000,B 0.000,C 90.000,E1 5.853} C_DIS
LIN {X 0.045,Y -466.230,Z 476.817,A 0.000,B 0.000,C 90.000,E1 2.980} C_DIS
LIN {X -0.212,Y -467.501,Z 476.804,A 0.000,B 0.000,C 90.000,E1 0.802} C_DIS
LIN {X -0.043,Y -469.599,Z 476.790,A 0.000,B 0.000,C 90.000,E1 358.224} C_DIS
LIN {X 0.087,Y -472.154,Z 476.776,A 0.000,B 0.000,C 90.000,E1 355.698} C_DIS
LIN {X -0.124,Y -475.205,Z 476.762,A 0.000,B 0.000,C 90.000,E1 353.223} C_DIS
LIN {X 0.021,Y -478.176,Z 476.750,A 0.000,B 0.000,C 90.000,E1 351.027} C_DIS
LIN {X 0.120,Y -482.505,Z 476.735,A 0.000,B 0.000,C 90.000,E1 348.229} C_DIS
LIN {X -0.136,Y -489.600,Z 476.714,A 0.000,B 0.000,C 90.000,E1 344.574} C_DIS
LIN {X 0.082,Y -494.307,Z 476.702,A 0.000,B 0.000,C 90.000,E1 342.417} C_DIS
LIN {X 0.057,Y -498.506,Z 476.692,A 0.000,B 0.000,C 90.000,E1 340.604} C_DIS
LIN {X -0.100,Y -503.537,Z 476.681,A 0.000,B 0.000,C 90.000,E1 338.518} C_DIS
LIN {X 0.140,Y -507.084,Z 476.672,A 0.000,B 0.000,C 90.000,E1 336.997} C_DIS
LIN {X -0.097,Y -510.522,Z 476.664,A 0.000,B 0.000,C 90.000,E1 335.537} C_DIS
LIN {X -0.032,Y -515.327,Z 476.653,A 0.000,B 0.000,C 90.000,E1 333.461} C_DIS
LIN {X 0.150,Y -520.038,Z 476.641,A 0.000,B 0.000,C 90.000,E1 331.385} C_DIS
LIN {X 0.261,Y -524.908,Z 476.630,A 0.000,B 0.000,C 90.000,E1 329.331} C_DIS
LIN {X 0.075,Y -529.207,Z 476.620,A 0.000,B 0.000,C 90.000,E1 327.612} C_DIS
LIN {X 0.095,Y -533.525,Z 476.611,A 0.000,B 0.000,C 90.000,E1 325.881} C_DIS
LIN {X -0.227,Y -537.160,Z 476.603,A 0.000,B 0.000,C 90.000,E1 324.482} C_DIS
LIN {X -0.126,Y -542.364,Z 476.592,A 0.000,B 0.000,C 90.000,E1 322.477} C_DIS
LIN {X 0.023,Y -546.015,Z 476.584,A 0.000,B 0.000,C 90.000,E1 321.045} C_DIS
LIN {X -0.220,Y -550.446,Z 476.574,A 0.000,B 0.000,C 90.000,E1 319.380} C_DIS
LIN {X 0.005,Y -554.717,Z 476.565,A 0.000,B 0.000,C 90.000,E1 317.676} C_DIS
LIN {X 0.326,Y -558.976,Z 476.556,A 0.000,B 0.000,C 90.000,E1 315.972} C_DIS
LIN {X -0.008,Y -563.736,Z 476.545,A 0.000,B 0.000,C 90.000,E1 314.069} C_DIS
LIN {X 0.011,Y -567.185,Z 476.537,A 0.000,B 0.000,C 90.000,E1 312.690} C_DIS
LIN {X 0.105,Y -570.606,Z 476.530,A 0.000,B 0.000,C 90.000,E1 311.310} C_DIS
LIN {X 0.094,Y -575.257,Z 476.519,A 0.000,B 0.000,C 90.000,E1 309.402} C_DIS
LIN {X 0.042,Y -578.624,Z 476.511,A 0.000,B 0.000,C 90.000,E1 308.051} C_DIS
LIN {X -0.051,Y -581.979,Z 476.504,A 0.000,B 0.000,C 90.000,E1 306.710} C_DIS
LIN {X -0.137,Y -585.961,Z 476.495,A 0.000,B 0.000,C 90.000,E1 305.105} C_DIS
LIN {X -0.331,Y -589.251,Z 476.488,A 0.000,B 0.000,C 90.000,E1 303.785} C_DIS
LIN {X 0.022,Y -592.471,Z 476.480,A 0.000,B 0.000,C 90.000,E1 302.418} C_DIS
LIN {X 0.220,Y -594.906,Z 476.474,A 0.000,B 0.000,C 90.000,E1 301.337} C_DIS
LIN {X -0.368,Y -597.137,Z 476.468,A 0.000,B 0.000,C 90.000,E1 300.335} C_DIS
LIN {X -0.201,Y -599.748,Z 476.461,A 0.000,B 0.000,C 90.000,E1 298.999} C_DIS
LIN {X 0.244,Y -602.183,Z 476.454,A 0.000,B 0.000,C 90.000,E1 297.641} C_DIS
LIN {X -0.015,Y -603.979,Z 476.448,A 0.000,B 0.000,C 90.000,E1 296.616} C_DIS
LIN {X -0.251,Y -605.561,Z 476.442,A 0.000,B 0.000,C 90.000,E1 295.591} C_DIS
LIN {X 0.078,Y -606.939,Z 476.436,A 0.000,B 0.000,C 90.000,E1 294.515} C_DIS
LIN {X 0.131,Y -608.453,Z 476.429,A 0.000,B 0.000,C 90.000,E1 293.206} C_DIS
LIN {X -0.068,Y -610.235,Z 476.420,A 0.000,B 0.000,C 90.000,E1 291.663} C_DIS
LIN {X -0.233,Y -611.746,Z 476.412,A 0.000,B 0.000,C 90.000,E1 290.120} C_DIS
LIN {X 0.244,Y -612.903,Z 476.405,A 0.000,B 0.000,C 90.000,E1 288.779} C_DIS
LIN {X -0.289,Y -614.232,Z 476.396,A 0.000,B 0.000,C 90.000,E1 287.275} C_DIS
LIN {X -0.141,Y -615.178,Z 476.389,A 0.000,B 0.000,C 90.000,E1 285.969} C_DIS
LIN {X -0.049,Y -616.155,Z 476.380,A 0.000,B 0.000,C 90.000,E1 284.411} C_DIS
LIN {X -0.024,Y -616.728,Z 476.373,A 0.000,B 0.000,C 90.000,E1 283.119} C_DIS
LIN {X 0.016,Y -617.263,Z 476.366,A 0.000,B 0.000,C 90.000,E1 281.827} C_DIS
LIN {X -0.200,Y -617.402,Z 476.361,A 0.000,B 0.000,C 90.000,E1 281.074} C_DIS
LIN {X -0.161,Y -617.562,Z 476.354,A 0.000,B 0.000,C 90.000,E1 279.782} C_DIS
LIN {X 0.274,Y -617.424,Z 476.347,A 0.000,B 0.000,C 90.000,E1 278.454} C_DIS
LIN {X -0.178,Y -617.111,Z 476.341,A 0.000,B 0.000,C 90.000,E1 277.466} C_DIS
LIN {X 0.181,Y -616.521,Z 476.334,A 0.000,B 0.000,C 90.000,E1 276.144} C_DIS
LIN {X -0.044,Y -616.031,Z 476.330,A 0.000,B 0.000,C 90.000,E1 275.391} C_DIS
LIN {X 0.252,Y -614.873,Z 476.323,A 0.000,B 0.000,C 90.000,E1 274.073} C_DIS
LIN {X -0.047,Y -614.012,Z 476.319,A 0.000,B 0.000,C 90.000,E1 273.326} C_DIS
LIN {X 0.229,Y -612.358,Z 476.311,A 0.000,B 0.000,C 90.000,E1 272.007} C_DIS
LIN {X -0.106,Y -611.225,Z 476.307,A 0.000,B 0.000,C 90.000,E1 271.260} C_DIS
LIN {X -0.228,Y -608.732,Z 476.298,A 0.000,B 0.000,C 90.000,E1 269.714} C_DIS
LIN {X -0.069,Y -606.402,Z 476.291,A 0.000,B 0.000,C 90.000,E1 268.396} C_DIS
LIN {X -0.196,Y -604.508,Z 476.285,A 0.000,B 0.000,C 90.000,E1 267.364} C_DIS
LIN {X -0.098,Y -601.907,Z 476.278,A 0.000,B 0.000,C 90.000,E1 266.045} C_DIS
LIN {X -0.006,Y -599.168,Z 476.271,A 0.000,B 0.000,C 90.000,E1 264.723} C_DIS
LIN {X -0.277,Y -595.643,Z 476.262,A 0.000,B 0.000,C 90.000,E1 263.166} C_DIS
LIN {X -0.225,Y -592.659,Z 476.255,A 0.000,B 0.000,C 90.000,E1 261.837} C_DIS
LIN {X 0.129,Y -589.012,Z 476.246,A 0.000,B 0.000,C 90.000,E1 260.208} C_DIS
LIN {X -0.168,Y -585.097,Z 476.237,A 0.000,B 0.000,C 90.000,E1 258.634} C_DIS
LIN {X 0.143,Y -581.056,Z 476.228,A 0.000,B 0.000,C 90.000,E1 256.992} C_DIS
LIN {X 0.137,Y -577.636,Z 476.220,A 0.000,B 0.000,C 90.000,E1 255.644} C_DIS
LIN {X 0.004,Y -573.336,Z 476.211,A 0.000,B 0.000,C 90.000,E1 254.031} C_DIS
LIN {X -0.184,Y -570.407,Z 476.205,A 0.000,B 0.000,C 90.000,E1 252.960} C_DIS
LIN {X 0.296,Y -567.393,Z 476.199,A 0.000,B 0.000,C 90.000,E1 251.819} C_DIS
LIN {X -0.016,Y -563.418,Z 476.192,A 0.000,B 0.000,C 90.000,E1 250.477} C_DIS
LIN {X 0.135,Y -559.284,Z 476.184,A 0.000,B 0.000,C 90.000,E1 249.082} C_DIS
LIN {X 0.106,Y -555.842,Z 476.178,A 0.000,B 0.000,C 90.000,E1 247.975} C_DIS
LIN {X -0.205,Y -551.332,Z 476.170,A 0.000,B 0.000,C 90.000,E1 246.613} C_DIS
LIN {X -0.134,Y -547.570,Z 476.164,A 0.000,B 0.000,C 90.000,E1 245.485} C_DIS
LIN {X -0.137,Y -542.727,Z 476.156,A 0.000,B 0.000,C 90.000,E1 244.076} C_DIS
LIN {X -0.009,Y -536.892,Z 476.146,A 0.000,B 0.000,C 90.000,E1 242.359} C_DIS
LIN {X 0.044,Y -532.023,Z 476.139,A 0.000,B 0.000,C 90.000,E1 240.923} C_DIS
LIN {X -0.076,Y -525.194,Z 476.127,A 0.000,B 0.000,C 90.000,E1 238.918} C_DIS
LIN {X -0.027,Y -519.394,Z 476.118,A 0.000,B 0.000,C 90.000,E1 237.168} C_DIS
LIN {X 0.237,Y -514.468,Z 476.109,A 0.000,B 0.000,C 90.000,E1 235.674} C_DIS
LIN {X 0.268,Y -509.312,Z 476.101,A 0.000,B 0.000,C 90.000,E1 234.196} C_DIS
LIN {X -0.177,Y -498.500,Z 476.083,A 0.000,B 0.000,C 90.000,E1 230.964} C_DIS
LIN {X -0.187,Y -492.261,Z 476.071,A 0.000,B 0.000,C 90.000,E1 228.852} C_DIS
LIN {X 0.144,Y -487.036,Z 476.061,A 0.000,B 0.000,C 90.000,E1 226.986} C_DIS
LIN {X 0.001,Y -481.904,Z 476.051,A 0.000,B 0.000,C 90.000,E1 225.162} C_DIS
LIN {X -0.138,Y -476.182,Z 476.039,A 0.000,B 0.000,C 90.000,E1 223.014} C_DIS
LIN {X 0.045,Y -470.040,Z 476.025,A 0.000,B 0.000,C 90.000,E1 220.496} C_DIS
LIN {X -0.028,Y -465.025,Z 476.013,A 0.000,B 0.000,C 90.000,E1 218.302} C_DIS
LIN {X -0.087,Y -460.333,Z 476.000,A 0.000,B 0.000,C 90.000,E1 216.091} C_DIS
LIN {X 0.098,Y -455.839,Z 475.988,A 0.000,B 0.000,C 90.000,E1 213.833} C_DIS
LIN {X 0.028,Y -451.519,Z 475.976,A 0.000,B 0.000,C 90.000,E1 211.592} C_DIS
LIN {X -0.241,Y -449.116,Z 475.968,A 0.000,B 0.000,C 90.000,E1 210.335} C_DIS
LIN {X 0.048,Y -444.934,Z 475.956,A 0.000,B 0.000,C 90.000,E1 208.025} C_DIS
LIN {X -0.092,Y -441.930,Z 475.947,A 0.000,B 0.000,C 90.000,E1 206.411} C_DIS
LIN {X -0.247,Y -438.275,Z 475.936,A 0.000,B 0.000,C 90.000,E1 204.463} C_DIS
LIN {X -0.078,Y -434.613,Z 475.925,A 0.000,B 0.000,C 90.000,E1 202.461} C_DIS
LIN {X 0.076,Y -429.377,Z 475.908,A 0.000,B 0.000,C 90.000,E1 199.450} C_DIS
LIN {X -0.033,Y -426.127,Z 475.897,A 0.000,B 0.000,C 90.000,E1 197.457} C_DIS
LIN {X -0.096,Y -422.195,Z 475.882,A 0.000,B 0.000,C 90.000,E1 194.773} C_DIS
LIN {X 0.105,Y -419.541,Z 475.871,A 0.000,B 0.000,C 90.000,E1 192.715} C_DIS
LIN {X -0.007,Y -415.832,Z 475.854,A 0.000,B 0.000,C 90.000,E1 189.670} C_DIS
LIN {X -0.108,Y -412.803,Z 475.839,A 0.000,B 0.000,C 90.000,E1 186.947} C_DIS
LIN {X -0.034,Y -411.098,Z 475.829,A 0.000,B 0.000,C 90.000,E1 185.220} C_DIS
LIN {X -0.038,Y -408.631,Z 475.814,A 0.000,B 0.000,C 90.000,E1 182.465} C_DIS
LIN {X -0.167,Y -406.455,Z 475.796,A 0.000,B 0.000,C 90.000,E1 179.370} C_DIS
LIN {X 0.046,Y -404.988,Z 475.779,A 0.000,B 0.000,C 90.000,E1 176.216} C_DIS
LIN {X -0.114,Y -404.231,Z 475.762,A 0.000,B 0.000,C 90.000,E1 173.109} C_DIS
LIN {X -0.152,Y -404.246,Z 475.748,A 0.000,B 0.000,C 90.000,E1 170.679} C_DIS
LIN {X -0.051,Y -404.756,Z 475.735,A 0.000,B 0.000,C 90.000,E1 168.229} C_DIS
LIN {X -0.152,Y -405.692,Z 475.721,A 0.000,B 0.000,C 90.000,E1 165.811} C_DIS
LIN {X 0.056,Y -406.392,Z 475.713,A 0.000,B 0.000,C 90.000,E1 164.393} C_DIS
LIN {X 0.059,Y -408.410,Z 475.696,A 0.000,B 0.000,C 90.000,E1 161.275} C_DIS
LIN {X 0.153,Y -411.078,Z 475.679,A 0.000,B 0.000,C 90.000,E1 158.156} C_DIS
LIN {X -0.158,Y -413.489,Z 475.665,A 0.000,B 0.000,C 90.000,E1 155.793} C_DIS
LIN {X -0.001,Y -415.731,Z 475.654,A 0.000,B 0.000,C 90.000,E1 153.717} C_DIS
LIN {X 0.159,Y -418.495,Z 475.641,A 0.000,B 0.000,C 90.000,E1 151.307} C_DIS
LIN {X 0.105,Y -420.459,Z 475.631,A 0.000,B 0.000,C 90.000,E1 149.616} C_DIS
LIN {X 0.154,Y -422.391,Z 475.622,A 0.000,B 0.000,C 90.000,E1 147.916} C_DIS
LIN {X 0.040,Y -423.975,Z 475.614,A 0.000,B 0.000,C 90.000,E1 146.580} C_DIS
LIN {X 0.022,Y -426.407,Z 475.603,A 0.000,B 0.000,C 90.000,E1 144.562} C_DIS
LIN {X -0.012,Y -428.433,Z 475.594,A 0.000,B 0.000,C 90.000,E1 142.889} C_DIS
LIN {X -0.016,Y -430.993,Z 475.583,A 0.000,B 0.000,C 90.000,E1 140.884} C_DIS
LIN {X 0.055,Y -432.669,Z 475.575,A 0.000,B 0.000,C 90.000,E1 139.542} C_DIS
LIN {X 0.026,Y -435.044,Z 475.564,A 0.000,B 0.000,C 90.000,E1 137.553} C_DIS
LIN {X -0.086,Y -435.850,Z 475.561,A 0.000,B 0.000,C 90.000,E1 136.905} C_DIS
LIN {X 0.028,Y -437.051,Z 475.553,A 0.000,B 0.000,C 90.000,E1 135.567} C_DIS
LIN {X -0.110,Y -437.845,Z 475.548,A 0.000,B 0.000,C 90.000,E1 134.595} C_DIS
LIN {X 0.036,Y -438.543,Z 475.540,A 0.000,B 0.000,C 90.000,E1 133.257} C_DIS
LIN {X 0.194,Y -438.991,Z 475.533,A 0.000,B 0.000,C 90.000,E1 131.919} C_DIS
LIN {X 0.059,Y -438.755,Z 475.526,A 0.000,B 0.000,C 90.000,E1 130.620} C_DIS
LIN {X -0.034,Y -438.122,Z 475.520,A 0.000,B 0.000,C 90.000,E1 129.644} C_DIS
LIN {X -0.135,Y -437.292,Z 475.515,A 0.000,B 0.000,C 90.000,E1 128.669} C_DIS
LIN {X 0.103,Y -435.720,Z 475.507,A 0.000,B 0.000,C 90.000,E1 127.317} C_DIS
LIN {X -0.039,Y -434.318,Z 475.502,A 0.000,B 0.000,C 90.000,E1 126.343} C_DIS
LIN {X -0.103,Y -432.188,Z 475.495,A 0.000,B 0.000,C 90.000,E1 125.025} C_DIS
LIN {X -0.195,Y -429.708,Z 475.487,A 0.000,B 0.000,C 90.000,E1 123.706} C_DIS
LIN {X 0.030,Y -427.085,Z 475.480,A 0.000,B 0.000,C 90.000,E1 122.339} C_DIS
LIN {X -0.160,Y -426.055,Z 475.477,A 0.000,B 0.000,C 90.000,E1 121.878} C_DIS
LIN {X -0.198,Y -426.052,Z 475.477,A 0.000,B 0.000,C 90.000,E1 121.878} C_DIS
LIN {X -0.023,Y -430.633,Z 475.469,A 0.000,B 0.000,C 90.000,E1 120.335} C_DIS
LIN {X -0.030,Y -441.537,Z 475.445,A 0.000,B 0.000,C 90.000,E1 116.027} C_DIS
LIN {X 0.097,Y -444.453,Z 475.439,A 0.000,B 0.000,C 90.000,E1 115.027} C_DIS
LIN {X -0.004,Y -445.924,Z 475.436,A 0.000,B 0.000,C 90.000,E1 114.387} C_DIS
LIN {X 0.133,Y -455.330,Z 475.414,A 0.000,B 0.000,C 90.000,E1 110.482} C_DIS
LIN {X -0.072,Y -457.131,Z 475.410,A 0.000,B 0.000,C 90.000,E1 109.866} C_DIS
LIN {X -0.224,Y -466.529,Z 475.386,A 0.000,B 0.000,C 90.000,E1 105.426} C_DIS
LIN {X -0.047,Y -467.988,Z 475.382,A 0.000,B 0.000,C 90.000,E1 104.773} C_DIS
LIN {X -0.100,Y -473.525,Z 475.363,A 0.000,B 0.000,C 90.000,E1 101.422} C_DIS
LIN {X -0.138,Y -503.391,Z 475.363,A 0.000,B 0.000,C 90.000,E1 101.422} C_DIS
LIN {X 0.115,Y -513.733,Z 475.363,A 0.000,B 0.000,C 90.000,E1 101.366} C_DIS
LIN {X -0.262,Y -519.677,Z 475.363,A 0.000,B 0.000,C 90.000,E1 101.366} C_DIS
LIN {X -0.238,Y -530.085,Z 475.362,A 0.000,B 0.000,C 90.000,E1 101.243} C_DIS
LIN {X -0.128,Y -536.446,Z 475.362,A 0.000,B 0.000,C 90.000,E1 101.130} C_DIS
LIN {X -0.233,Y -543.293,Z 475.361,A 0.000,B 0.000,C 90.000,E1 101.007} C_DIS
LIN {X -0.086,Y -549.739,Z 475.360,A 0.000,B 0.000,C 90.000,E1 100.838} C_DIS
LIN {X -0.167,Y -556.619,Z 475.359,A 0.000,B 0.000,C 90.000,E1 100.658} C_DIS
LIN {X 0.033,Y -563.191,Z 475.358,A 0.000,B 0.000,C 90.000,E1 100.433} C_DIS
LIN {X 0.041,Y -569.708,Z 475.357,A 0.000,B 0.000,C 90.000,E1 100.197} C_DIS
LIN {X 0.202,Y -579.632,Z 475.355,A 0.000,B 0.000,C 90.000,E1 99.792} C_DIS
LIN {X 0.057,Y -587.541,Z 475.353,A 0.000,B 0.000,C 90.000,E1 99.443} C_DIS
LIN {X -0.071,Y -589.145,Z 475.352,A 0.000,B 0.000,C 90.000,E1 99.378} C_DIS
LIN {X 0.114,Y -598.202,Z 475.349,A 0.000,B 0.000,C 90.000,E1 98.859} C_DIS
LIN {X 0.116,Y -601.188,Z 475.348,A 0.000,B 0.000,C 90.000,E1 98.681} C_DIS
LIN {X -0.203,Y -606.662,Z 475.346,A 0.000,B 0.000,C 90.000,E1 98.341} C_DIS
LIN {X 0.195,Y -610.775,Z 475.345,A 0.000,B 0.000,C 90.000,E1 97.992} C_DIS
LIN {X 0.309,Y -612.430,Z 475.344,A 0.000,B 0.000,C 90.000,E1 97.871} C_DIS
LIN {X -0.142,Y -619.934,Z 475.340,A 0.000,B 0.000,C 90.000,E1 97.239} C_DIS
LIN {X 0.143,Y -624.850,Z 475.337,A 0.000,B 0.000,C 90.000,E1 96.720} C_DIS
LIN {X 0.113,Y -631.283,Z 475.333,A 0.000,B 0.000,C 90.000,E1 95.967} C_DIS
LIN {X 0.110,Y -635.591,Z 475.330,A 0.000,B 0.000,C 90.000,E1 95.334} C_DIS
LIN {X 0.142,Y -639.446,Z 475.326,A 0.000,B 0.000,C 90.000,E1 94.702} C_DIS
LIN {X 0.085,Y -643.370,Z 475.322,A 0.000,B 0.000,C 90.000,E1 93.955} C_DIS
LIN {X 0.254,Y -645.634,Z 475.319,A 0.000,B 0.000,C 90.000,E1 93.440} C_DIS
LIN {X -0.170,Y -647.580,Z 475.317,A 0.000,B 0.000,C 90.000,E1 92.980} C_DIS
LIN {X -0.185,Y -649.759,Z 475.312,A 0.000,B 0.000,C 90.000,E1 92.236} C_DIS
LIN {X 0.059,Y -650.909,Z 475.310,A 0.000,B 0.000,C 90.000,E1 91.718} C_DIS
LIN {X 0.289,Y -651.738,Z 475.307,A 0.000,B 0.000,C 90.000,E1 91.203} C_DIS
LIN {X -0.126,Y -652.268,Z 475.304,A 0.000,B 0.000,C 90.000,E1 90.745} C_DIS
LIN {X -0.086,Y -652.475,Z 475.300,A 0.000,B 0.000,C 90.000,E1 90.000} C_DIS
LIN {X 0.160,Y -652.224,Z 475.297,A 0.000,B 0.000,C 90.000,E1 89.484} C_DIS
LIN {X -0.248,Y -651.765,Z 475.295,A 0.000,B 0.000,C 90.000,E1 89.026} C_DIS
LIN {X -0.217,Y -650.440,Z 475.290,A 0.000,B 0.000,C 90.000,E1 88.282} C_DIS
LIN {X 0.035,Y -649.293,Z 475.288,A 0.000,B 0.000,C 90.000,E1 87.764} C_DIS
LIN {X 0.255,Y -647.696,Z 475.285,A 0.000,B 0.000,C 90.000,E1 87.249} C_DIS
LIN {X 0.271,Y -644.743,Z 475.281,A 0.000,B 0.000,C 90.000,E1 86.502} C_DIS
LIN {X -0.261,Y -641.663,Z 475.277,A 0.000,B 0.000,C 90.000,E1 85.927} C_DIS
LIN {X 0.080,Y -635.672,Z 475.272,A 0.000,B 0.000,C 90.000,E1 84.894} C_DIS
LIN {X -0.030,Y -630.173,Z 475.268,A 0.000,B 0.000,C 90.000,E1 84.147} C_DIS
LIN {X -0.050,Y -625.209,Z 475.264,A 0.000,B 0.000,C 90.000,E1 83.514} C_DIS
LIN {X -0.040,Y -619.467,Z 475.260,A 0.000,B 0.000,C 90.000,E1 82.875} C_DIS
LIN {X -0.039,Y -613.202,Z 475.257,A 0.000,B 0.000,C 90.000,E1 82.243} C_DIS
LIN {X 0.225,Y -607.782,Z 475.254,A 0.000,B 0.000,C 90.000,E1 81.724} C_DIS
LIN {X -0.268,Y -599.233,Z 475.250,A 0.000,B 0.000,C 90.000,E1 81.084} C_DIS
LIN {X -0.113,Y -594.888,Z 475.249,A 0.000,B 0.000,C 90.000,E1 80.735} C_DIS
LIN {X 0.186,Y -590.188,Z 475.247,A 0.000,B 0.000,C 90.000,E1 80.387} C_DIS
LIN {X -0.256,Y -583.821,Z 475.245,A 0.000,B 0.000,C 90.000,E1 80.038} C_DIS
LIN {X -0.069,Y -578.563,Z 475.243,A 0.000,B 0.000,C 90.000,E1 79.746} C_DIS
LIN {X 0.172,Y -571.698,Z 475.241,A 0.000,B 0.000,C 90.000,E1 79.398} C_DIS
LIN {X -0.043,Y -565.876,Z 475.240,A 0.000,B 0.000,C 90.000,E1 79.218} C_DIS
LIN {X -0.007,Y -559.565,Z 475.239,A 0.000,B 0.000,C 90.000,E1 79.050} C_DIS
LIN {X 0.062,Y -552.998,Z 475.239,A 0.000,B 0.000,C 90.000,E1 78.926} C_DIS
LIN {X 0.076,Y -546.361,Z 475.238,A 0.000,B 0.000,C 90.000,E1 78.870} C_DIS
LIN {X 0.041,Y -542.203,Z 475.238,A 0.000,B 0.000,C 90.000,E1 78.870} C_DIS
LIN {X 0.007,Y -481.902,Z 475.238,A 0.000,B 0.000,C 90.000,E1 78.870} C_DIS
LIN {X 0.052,Y -480.551,Z 475.227,A 0.000,B 0.000,C 90.000,E1 76.881} C_DIS
LIN {X -0.037,Y -474.306,Z 475.201,A 0.000,B 0.000,C 90.000,E1 72.236} C_DIS
LIN {X -0.216,Y -473.892,Z 475.200,A 0.000,B 0.000,C 90.000,E1 71.945} C_DIS
LIN {X -0.089,Y -466.285,Z 475.175,A 0.000,B 0.000,C 90.000,E1 67.539} C_DIS
LIN {X -0.145,Y -465.854,Z 475.173,A 0.000,B 0.000,C 90.000,E1 67.230} C_DIS
LIN {X -0.204,Y -465.283,Z 475.172,A 0.000,B 0.000,C 90.000,E1 66.922} C_DIS
LIN {X 0.172,Y -456.897,Z 475.149,A 0.000,B 0.000,C 90.000,E1 62.743} C_DIS
LIN {X 0.255,Y -455.528,Z 475.144,A 0.000,B 0.000,C 90.000,E1 61.897} C_DIS
LIN {X 0.216,Y -455.544,Z 475.144,A 0.000,B 0.000,C 90.000,E1 61.897} C_DIS
LIN {X 0.022,Y -461.149,Z 475.139,A 0.000,B 0.000,C 90.000,E1 61.001} C_DIS
LIN {X 0.013,Y -466.701,Z 475.134,A 0.000,B 0.000,C 90.000,E1 60.049} C_DIS
LIN {X -0.162,Y -471.026,Z 475.129,A 0.000,B 0.000,C 90.000,E1 59.282} C_DIS
LIN {X 0.188,Y -475.028,Z 475.125,A 0.000,B 0.000,C 90.000,E1 58.456} C_DIS
LIN {X -0.283,Y -476.592,Z 475.123,A 0.000,B 0.000,C 90.000,E1 58.201} C_DIS
LIN {X 0.125,Y -479.902,Z 475.119,A 0.000,B 0.000,C 90.000,E1 57.375} C_DIS
LIN {X 0.132,Y -482.267,Z 475.115,A 0.000,B 0.000,C 90.000,E1 56.755} C_DIS
LIN {X -0.112,Y -484.170,Z 475.112,A 0.000,B 0.000,C 90.000,E1 56.167} C_DIS
LIN {X -0.078,Y -485.804,Z 475.109,A 0.000,B 0.000,C 90.000,E1 55.548} C_DIS
LIN {X 0.021,Y -486.586,Z 475.107,A 0.000,B 0.000,C 90.000,E1 55.229} C_DIS
LIN {X -0.090,Y -488.398,Z 475.102,A 0.000,B 0.000,C 90.000,E1 54.322} C_DIS
LIN {X -0.023,Y -489.424,Z 475.098,A 0.000,B 0.000,C 90.000,E1 53.703} C_DIS
LIN {X 0.183,Y -490.518,Z 475.093,A 0.000,B 0.000,C 90.000,E1 52.763} C_DIS
LIN {X -0.286,Y -491.309,Z 475.088,A 0.000,B 0.000,C 90.000,E1 51.904} C_DIS
LIN {X -0.060,Y -491.865,Z 475.083,A 0.000,B 0.000,C 90.000,E1 50.964} C_DIS
LIN {X -0.048,Y -492.302,Z 475.076,A 0.000,B 0.000,C 90.000,E1 49.747} C_DIS
LIN {X -0.193,Y -492.499,Z 475.071,A 0.000,B 0.000,C 90.000,E1 48.852} C_DIS
LIN {X -0.010,Y -492.556,Z 475.066,A 0.000,B 0.000,C 90.000,E1 47.919} C_DIS
LIN {X 0.012,Y -492.427,Z 475.060,A 0.000,B 0.000,C 90.000,E1 46.701} C_DIS
LIN {X -0.165,Y -492.248,Z 475.054,A 0.000,B 0.000,C 90.000,E1 45.810} C_DIS
LIN {X 0.005,Y -491.747,Z 475.046,A 0.000,B 0.000,C 90.000,E1 44.271} C_DIS
LIN {X -0.011,Y -491.188,Z 475.039,A 0.000,B 0.000,C 90.000,E1 43.056} C_DIS
LIN {X 0.150,Y -490.231,Z 475.031,A 0.000,B 0.000,C 90.000,E1 41.515} C_DIS
LIN {X -0.029,Y -489.161,Z 475.022,A 0.000,B 0.000,C 90.000,E1 40.011} C_DIS
LIN {X 0.150,Y -488.045,Z 475.014,A 0.000,B 0.000,C 90.000,E1 38.463} C_DIS
LIN {X 0.009,Y -486.863,Z 475.005,A 0.000,B 0.000,C 90.000,E1 36.950} C_DIS
LIN {X 0.014,Y -485.826,Z 474.999,A 0.000,B 0.000,C 90.000,E1 35.724} C_DIS
LIN {X -0.063,Y -484.415,Z 474.990,A 0.000,B 0.000,C 90.000,E1 34.199} C_DIS
LIN {X -0.166,Y -482.816,Z 474.981,A 0.000,B 0.000,C 90.000,E1 32.673} C_DIS
LIN {X -0.156,Y -481.120,Z 474.973,A 0.000,B 0.000,C 90.000,E1 31.131} C_DIS
LIN {X 0.237,Y -479.353,Z 474.964,A 0.000,B 0.000,C 90.000,E1 29.539} C_DIS
LIN {X -0.092,Y -477.188,Z 474.954,A 0.000,B 0.000,C 90.000,E1 27.719} C_DIS
LIN {X -0.046,Y -475.171,Z 474.944,A 0.000,B 0.000,C 90.000,E1 25.848} C_DIS
LIN {X 0.070,Y -472.589,Z 474.928,A 0.000,B 0.000,C 90.000,E1 23.025} C_DIS
LIN {X -0.010,Y -471.005,Z 474.916,A 0.000,B 0.000,C 90.000,E1 20.844} C_DIS
LIN {X 0.099,Y -470.261,Z 474.909,A 0.000,B 0.000,C 90.000,E1 19.577} C_DIS
LIN {X 0.102,Y -469.148,Z 474.898,A 0.000,B 0.000,C 90.000,E1 17.692} C_DIS
LIN {X -0.014,Y -468.265,Z 474.890,A 0.000,B 0.000,C 90.000,E1 16.134} C_DIS
LIN {X 0.171,Y -467.003,Z 474.876,A 0.000,B 0.000,C 90.000,E1 13.592} C_DIS
LIN {X -0.073,Y -466.120,Z 474.860,A 0.000,B 0.000,C 90.000,E1 10.782} C_DIS
LIN {X -0.048,Y -465.713,Z 474.844,A 0.000,B 0.000,C 90.000,E1 7.936} C_DIS
LIN {X 0.090,Y -466.094,Z 474.827,A 0.000,B 0.000,C 90.000,E1 4.759} C_DIS
LIN {X 0.075,Y -467.802,Z 474.806,A 0.000,B 0.000,C 90.000,E1 0.974} C_DIS
LIN {X 0.222,Y -470.301,Z 474.788,A 0.000,B 0.000,C 90.000,E1 357.879} C_DIS
LIN {X -0.057,Y -473.664,Z 474.771,A 0.000,B 0.000,C 90.000,E1 354.780} C_DIS
LIN {X -0.014,Y -476.395,Z 474.759,A 0.000,B 0.000,C 90.000,E1 352.591} C_DIS
LIN {X 0.084,Y -479.934,Z 474.745,A 0.000,B 0.000,C 90.000,E1 350.095} C_DIS
LIN {X -0.228,Y -484.501,Z 474.730,A 0.000,B 0.000,C 90.000,E1 347.353} C_DIS
LIN {X -0.060,Y -489.999,Z 474.714,A 0.000,B 0.000,C 90.000,E1 344.574} C_DIS
LIN {X 0.170,Y -494.736,Z 474.702,A 0.000,B 0.000,C 90.000,E1 342.417} C_DIS
LIN {X 0.155,Y -498.962,Z 474.692,A 0.000,B 0.000,C 90.000,E1 340.604} C_DIS
LIN {X -0.172,Y -504.054,Z 474.681,A 0.000,B 0.000,C 90.000,E1 338.539} C_DIS
LIN {X -0.205,Y -507.625,Z 474.672,A 0.000,B 0.000,C 90.000,E1 337.050} C_DIS
LIN {X 0.037,Y -511.090,Z 474.664,A 0.000,B 0.000,C 90.000,E1 335.537} C_DIS
LIN {X 0.118,Y -515.930,Z 474.653,A 0.000,B 0.000,C 90.000,E1 333.461} C_DIS
LIN {X -0.055,Y -520.056,Z 474.643,A 0.000,B 0.000,C 90.000,E1 331.719} C_DIS
LIN {X -0.271,Y -525.621,Z 474.630,A 0.000,B 0.000,C 90.000,E1 329.410} C_DIS
LIN {X -0.169,Y -529.951,Z 474.620,A 0.000,B 0.000,C 90.000,E1 327.661} C_DIS
LIN {X -0.125,Y -534.282,Z 474.611,A 0.000,B 0.000,C 90.000,E1 325.928} C_DIS
LIN {X 0.005,Y -537.221,Z 474.604,A 0.000,B 0.000,C 90.000,E1 324.769} C_DIS
LIN {X 0.108,Y -542.437,Z 474.593,A 0.000,B 0.000,C 90.000,E1 322.763} C_DIS
LIN {X -0.164,Y -546.149,Z 474.585,A 0.000,B 0.000,C 90.000,E1 321.376} C_DIS
LIN {X 0.027,Y -550.608,Z 474.576,A 0.000,B 0.000,C 90.000,E1 319.666} C_DIS
LIN {X -0.108,Y -554.929,Z 474.567,A 0.000,B 0.000,C 90.000,E1 318.000} C_DIS
LIN {X 0.213,Y -559.262,Z 474.557,A 0.000,B 0.000,C 90.000,E1 316.296} C_DIS
LIN {X -0.183,Y -563.389,Z 474.548,A 0.000,B 0.000,C 90.000,E1 314.676} C_DIS
LIN {X -0.087,Y -567.582,Z 474.539,A 0.000,B 0.000,C 90.000,E1 313.014} C_DIS
LIN {X 0.016,Y -571.070,Z 474.531,A 0.000,B 0.000,C 90.000,E1 311.634} C_DIS
LIN {X -0.117,Y -575.080,Z 474.522,A 0.000,B 0.000,C 90.000,E1 310.011} C_DIS
LIN {X 0.188,Y -578.547,Z 474.515,A 0.000,B 0.000,C 90.000,E1 308.624} C_DIS
LIN {X -0.082,Y -582.608,Z 474.506,A 0.000,B 0.000,C 90.000,E1 307.030} C_DIS
LIN {X 0.199,Y -586.632,Z 474.497,A 0.000,B 0.000,C 90.000,E1 305.391} C_DIS
LIN {X 0.020,Y -589.933,Z 474.489,A 0.000,B 0.000,C 90.000,E1 304.072} C_DIS
LIN {X -0.107,Y -593.175,Z 474.482,A 0.000,B 0.000,C 90.000,E1 302.752} C_DIS
LIN {X 0.099,Y -595.652,Z 474.476,A 0.000,B 0.000,C 90.000,E1 301.671} C_DIS
LIN {X 0.338,Y -597.951,Z 474.470,A 0.000,B 0.000,C 90.000,E1 300.590} C_DIS
LIN {X 0.228,Y -600.627,Z 474.463,A 0.000,B 0.000,C 90.000,E1 299.283} C_DIS
LIN {X 0.103,Y -603.557,Z 474.454,A 0.000,B 0.000,C 90.000,E1 297.719} C_DIS
LIN {X 0.138,Y -605.378,Z 474.448,A 0.000,B 0.000,C 90.000,E1 296.668} C_DIS
LIN {X -0.137,Y -607.392,Z 474.441,A 0.000,B 0.000,C 90.000,E1 295.387} C_DIS
LIN {X -0.038,Y -608.800,Z 474.435,A 0.000,B 0.000,C 90.000,E1 294.335} C_DIS
LIN {X 0.050,Y -610.357,Z 474.428,A 0.000,B 0.000,C 90.000,E1 293.025} C_DIS
LIN {X 0.165,Y -611.887,Z 474.421,A 0.000,B 0.000,C 90.000,E1 291.716} C_DIS
LIN {X 0.118,Y -612.961,Z 474.415,A 0.000,B 0.000,C 90.000,E1 290.684} C_DIS
LIN {X 0.048,Y -614.254,Z 474.408,A 0.000,B 0.000,C 90.000,E1 289.396} C_DIS
LIN {X -0.260,Y -615.633,Z 474.399,A 0.000,B 0.000,C 90.000,E1 287.873} C_DIS
LIN {X 0.083,Y -616.703,Z 474.392,A 0.000,B 0.000,C 90.000,E1 286.551} C_DIS
LIN {X 0.039,Y -617.842,Z 474.383,A 0.000,B 0.000,C 90.000,E1 285.009} C_DIS
LIN {X -0.277,Y -618.411,Z 474.378,A 0.000,B 0.000,C 90.000,E1 284.008} C_DIS
LIN {X 0.311,Y -619.147,Z 474.369,A 0.000,B 0.000,C 90.000,E1 282.411} C_DIS
LIN {X 0.264,Y -619.501,Z 474.362,A 0.000,B 0.000,C 90.000,E1 281.130} C_DIS
LIN {X 0.230,Y -619.690,Z 474.355,A 0.000,B 0.000,C 90.000,E1 279.849} C_DIS
LIN {X 0.194,Y -619.530,Z 474.348,A 0.000,B 0.000,C 90.000,E1 278.568} C_DIS
LIN {X -0.315,Y -619.269,Z 474.342,A 0.000,B 0.000,C 90.000,E1 277.587} C_DIS
LIN {X -0.138,Y -618.809,Z 474.336,A 0.000,B 0.000,C 90.000,E1 276.543} C_DIS
LIN {X -0.106,Y -618.235,Z 474.331,A 0.000,B 0.000,C 90.000,E1 275.511} C_DIS
LIN {X 0.285,Y -617.061,Z 474.323,A 0.000,B 0.000,C 90.000,E1 274.188} C_DIS
LIN {X -0.306,Y -615.881,Z 474.318,A 0.000,B 0.000,C 90.000,E1 273.212} C_DIS
LIN {X -0.296,Y -614.533,Z 474.312,A 0.000,B 0.000,C 90.000,E1 272.178} C_DIS
LIN {X 0.005,Y -613.381,Z 474.308,A 0.000,B 0.000,C 90.000,E1 271.375} C_DIS
LIN {X -0.075,Y -610.864,Z 474.299,A 0.000,B 0.000,C 90.000,E1 269.828} C_DIS
LIN {X -0.211,Y -608.007,Z 474.290,A 0.000,B 0.000,C 90.000,E1 268.282} C_DIS
LIN {X 0.288,Y -606.046,Z 474.285,A 0.000,B 0.000,C 90.000,E1 267.192} C_DIS
LIN {X -0.151,Y -603.387,Z 474.277,A 0.000,B 0.000,C 90.000,E1 265.927} C_DIS
LIN {X -0.077,Y -600.584,Z 474.270,A 0.000,B 0.000,C 90.000,E1 264.609} C_DIS
LIN {X -0.039,Y -596.394,Z 474.260,A 0.000,B 0.000,C 90.000,E1 262.761} C_DIS
LIN {X 0.025,Y -593.325,Z 474.252,A 0.000,B 0.000,C 90.000,E1 261.432} C_DIS
LIN {X 0.123,Y -590.168,Z 474.245,A 0.000,B 0.000,C 90.000,E1 260.095} C_DIS
LIN {X 0.166,Y -586.859,Z 474.238,A 0.000,B 0.000,C 90.000,E1 258.757} C_DIS
LIN {X 0.262,Y -583.424,Z 474.230,A 0.000,B 0.000,C 90.000,E1 257.409} C_DIS
LIN {X -0.045,Y -579.275,Z 474.221,A 0.000,B 0.000,C 90.000,E1 255.825} C_DIS
LIN {X 0.203,Y -575.651,Z 474.214,A 0.000,B 0.000,C 90.000,E1 254.448} C_DIS
LIN {X 0.047,Y -572.715,Z 474.208,A 0.000,B 0.000,C 90.000,E1 253.378} C_DIS
LIN {X 0.189,Y -568.931,Z 474.200,A 0.000,B 0.000,C 90.000,E1 252.000} C_DIS
LIN {X 0.106,Y -565.763,Z 474.194,A 0.000,B 0.000,C 90.000,E1 250.913} C_DIS
LIN {X 0.084,Y -560.843,Z 474.185,A 0.000,B 0.000,C 90.000,E1 249.263} C_DIS
LIN {X -0.134,Y -556.491,Z 474.177,A 0.000,B 0.000,C 90.000,E1 247.901} C_DIS
LIN {X 0.081,Y -551.910,Z 474.169,A 0.000,B 0.000,C 90.000,E1 246.485} C_DIS
LIN {X 0.158,Y -548.128,Z 474.163,A 0.000,B 0.000,C 90.000,E1 245.357} C_DIS
LIN {X -0.087,Y -542.261,Z 474.154,A 0.000,B 0.000,C 90.000,E1 243.691} C_DIS
LIN {X 0.027,Y -536.374,Z 474.144,A 0.000,B 0.000,C 90.000,E1 241.975} C_DIS
LIN {X -0.108,Y -532.475,Z 474.138,A 0.000,B 0.000,C 90.000,E1 240.845} C_DIS
LIN {X -0.031,Y -525.578,Z 474.127,A 0.000,B 0.000,C 90.000,E1 238.820} C_DIS
LIN {X -0.093,Y -520.744,Z 474.119,A 0.000,B 0.000,C 90.000,E1 237.375} C_DIS
LIN {X 0.197,Y -515.820,Z 474.111,A 0.000,B 0.000,C 90.000,E1 235.881} C_DIS
LIN {X -0.011,Y -512.795,Z 474.106,A 0.000,B 0.000,C 90.000,E1 235.022} C_DIS
LIN {X -0.001,Y -507.576,Z 474.098,A 0.000,B 0.000,C 90.000,E1 233.543} C_DIS
LIN {X -0.062,Y -497.940,Z 474.081,A 0.000,B 0.000,C 90.000,E1 230.561} C_DIS
LIN {X -0.077,Y -491.737,Z 474.069,A 0.000,B 0.000,C 90.000,E1 228.447} C_DIS
LIN {X 0.064,Y -485.650,Z 474.057,A 0.000,B 0.000,C 90.000,E1 226.296} C_DIS
LIN {X 0.224,Y -480.587,Z 474.047,A 0.000,B 0.000,C 90.000,E1 224.433} C_DIS
LIN {X -0.174,Y -474.160,Z 474.033,A 0.000,B 0.000,C 90.000,E1 222.000} C_DIS
LIN {X -0.130,Y -468.930,Z 474.021,A 0.000,B 0.000,C 90.000,E1 219.806} C_DIS
LIN {X -0.123,Y -463.313,Z 474.007,A 0.000,B 0.000,C 90.000,E1 217.282} C_DIS
LIN {X 0.142,Y -458.719,Z 473.995,A 0.000,B 0.000,C 90.000,E1 215.025} C_DIS
LIN {X 0.019,Y -454.293,Z 473.982,A 0.000,B 0.000,C 90.000,E1 212.801} C_DIS
LIN {X -0.031,Y -450.672,Z 473.972,A 0.000,B 0.000,C 90.000,E1 210.875} C_DIS
LIN {X -0.018,Y -445.846,Z 473.957,A 0.000,B 0.000,C 90.000,E1 208.281} C_DIS
LIN {X 0.105,Y -442.219,Z 473.946,A 0.000,B 0.000,C 90.000,E1 206.309} C_DIS
LIN {X 0.151,Y -438.545,Z 473.935,A 0.000,B 0.000,C 90.000,E1 204.335} C_DIS
LIN {X 0.149,Y -434.246,Z 473.923,A 0.000,B 0.000,C 90.000,E1 202.025} C_DIS
LIN {X -0.075,Y -429.598,Z 473.908,A 0.000,B 0.000,C 90.000,E1 199.396} C_DIS
LIN {X -0.173,Y -426.332,Z 473.897,A 0.000,B 0.000,C 90.000,E1 197.402} C_DIS
LIN {X 0.115,Y -422.859,Z 473.884,A 0.000,B 0.000,C 90.000,E1 195.009} C_DIS
LIN {X 0.080,Y -419.703,Z 473.870,A 0.000,B 0.000,C 90.000,E1 192.647} C_DIS
LIN {X -0.115,Y -415.999,Z 473.853,A 0.000,B 0.000,C 90.000,E1 189.613} C_DIS
LIN {X 0.164,Y -413.337,Z 473.840,A 0.000,B 0.000,C 90.000,E1 187.182} C_DIS
LIN {X -0.111,Y -410.596,Z 473.825,A 0.000,B 0.000,C 90.000,E1 184.473} C_DIS
LIN {X -0.135,Y -408.495,Z 473.811,A 0.000,B 0.000,C 90.000,E1 182.064} C_DIS
LIN {X 0.139,Y -406.405,Z 473.794,A 0.000,B 0.000,C 90.000,E1 178.912} C_DIS
LIN {X -0.029,Y -405.151,Z 473.779,A 0.000,B 0.000,C 90.000,E1 176.159} C_DIS
LIN {X -0.138,Y -404.475,Z 473.763,A 0.000,B 0.000,C 90.000,E1 173.394} C_DIS
LIN {X -0.215,Y -404.497,Z 473.746,A 0.000,B 0.000,C 90.000,E1 170.274} C_DIS
LIN {X -0.115,Y -404.988,Z 473.734,A 0.000,B 0.000,C 90.000,E1 168.173} C_DIS
LIN {X 0.180,Y -405.973,Z 473.721,A 0.000,B 0.000,C 90.000,E1 165.700} C_DIS
LIN {X -0.178,Y -407.252,Z 473.707,A 0.000,B 0.000,C 90.000,E1 163.323} C_DIS
LIN {X -0.144,Y -409.294,Z 473.692,A 0.000,B 0.000,C 90.000,E1 160.550} C_DIS
LIN {X 0.101,Y -411.459,Z 473.678,A 0.000,B 0.000,C 90.000,E1 158.103} C_DIS
LIN {X 0.044,Y -413.554,Z 473.667,A 0.000,B 0.000,C 90.000,E1 156.049} C_DIS
LIN {X 0.077,Y -415.430,Z 473.658,A 0.000,B 0.000,C 90.000,E1 154.332} C_DIS
LIN {X -0.151,Y -418.207,Z 473.644,A 0.000,B 0.000,C 90.000,E1 151.975} C_DIS
LIN {X 0.034,Y -419.809,Z 473.637,A 0.000,B 0.000,C 90.000,E1 150.589} C_DIS
LIN {X -0.113,Y -421.425,Z 473.629,A 0.000,B 0.000,C 90.000,E1 149.253} C_DIS
LIN {X 0.069,Y -423.821,Z 473.618,A 0.000,B 0.000,C 90.000,E1 147.199} C_DIS
LIN {X 0.027,Y -426.699,Z 473.605,A 0.000,B 0.000,C 90.000,E1 144.848} C_DIS
LIN {X -0.005,Y -428.839,Z 473.595,A 0.000,B 0.000,C 90.000,E1 143.176} C_DIS
LIN {X 0.005,Y -431.444,Z 473.584,A 0.000,B 0.000,C 90.000,E1 141.170} C_DIS
LIN {X 0.016,Y -433.657,Z 473.575,A 0.000,B 0.000,C 90.000,E1 139.504} C_DIS
LIN {X 0.021,Y -436.122,Z 473.564,A 0.000,B 0.000,C 90.000,E1 137.514} C_DIS
LIN {X -0.109,Y -437.324,Z 473.559,A 0.000,B 0.000,C 90.000,E1 136.539} C_DIS
LIN {X 0.023,Y -438.550,Z 473.551,A 0.000,B 0.000,C 90.000,E1 135.202} C_DIS
LIN {X 0.212,Y -439.293,Z 473.546,A 0.000,B 0.000,C 90.000,E1 134.190} C_DIS
LIN {X 0.060,Y -440.041,Z 473.538,A 0.000,B 0.000,C 90.000,E1 132.894} C_DIS
LIN {X -0.025,Y -440.354,Z 473.533,A 0.000,B 0.000,C 90.000,E1 131.919} C_DIS
LIN {X 0.189,Y -440.294,Z 473.527,A 0.000,B 0.000,C 90.000,E1 130.906} C_DIS
LIN {X -0.138,Y -440.252,Z 473.526,A 0.000,B 0.000,C 90.000,E1 130.620} C_DIS
LIN {X -0.213,Y -439.650,Z 473.520,A 0.000,B 0.000,C 90.000,E1 129.644} C_DIS
LIN {X 0.045,Y -438.847,Z 473.515,A 0.000,B 0.000,C 90.000,E1 128.624} C_DIS
LIN {X -0.033,Y -437.301,Z 473.507,A 0.000,B 0.000,C 90.000,E1 127.317} C_DIS
LIN {X 0.195,Y -435.882,Z 473.502,A 0.000,B 0.000,C 90.000,E1 126.297} C_DIS
LIN {X 0.145,Y -434.289,Z 473.496,A 0.000,B 0.000,C 90.000,E1 125.311} C_DIS
LIN {X 0.086,Y -431.836,Z 473.489,A 0.000,B 0.000,C 90.000,E1 123.992} C_DIS
LIN {X -0.015,Y -429.140,Z 473.482,A 0.000,B 0.000,C 90.000,E1 122.673} C_DIS
LIN {X -0.019,Y -426.832,Z 473.476,A 0.000,B 0.000,C 90.000,E1 121.592} C_DIS
LIN {X -0.058,Y -426.826,Z 473.476,A 0.000,B 0.000,C 90.000,E1 121.592} C_DIS
LIN {X -0.048,Y -430.644,Z 473.469,A 0.000,B 0.000,C 90.000,E1 120.335} C_DIS
LIN {X -0.055,Y -441.547,Z 473.445,A 0.000,B 0.000,C 90.000,E1 116.027} C_DIS
LIN {X 0.072,Y -444.464,Z 473.439,A 0.000,B 0.000,C 90.000,E1 115.027} C_DIS
LIN {X -0.029,Y -445.931,Z 473.436,A 0.000,B 0.000,C 90.000,E1 114.387} C_DIS
LIN {X 0.107,Y -455.340,Z 473.414,A 0.000,B 0.000,C 90.000,E1 110.482} C_DIS
LIN {X -0.097,Y -457.139,Z 473.410,A 0.000,B 0.000,C 90.000,E1 109.866} C_DIS
LIN {X 0.200,Y -466.537,Z 473.386,A 0.000,B 0.000,C 90.000,E1 105.371} C_DIS
LIN {X -0.074,Y -467.993,Z 473.382,A 0.000,B 0.000,C 90.000,E1 104.773} C_DIS
LIN {X 0.110,Y -474.508,Z 473.361,A 0.000,B 0.000,C 90.000,E1 100.894} C_DIS
LIN {X 0.072,Y -514.625,Z 473.361,A 0.000,B 0.000,C 90.000,E1 100.894} C_DIS
LIN {X -0.133,Y -526.916,Z 473.360,A 0.000,B 0.000,C 90.000,E1 100.838} C_DIS
LIN {X -0.277,Y -533.865,Z 473.360,A 0.000,B 0.000,C 90.000,E1 100.782} C_DIS
LIN {X 0.258,Y -541.471,Z 473.359,A 0.000,B 0.000,C 90.000,E1 100.602} C_DIS
LIN {X 0.040,Y -547.930,Z 473.358,A 0.000,B 0.000,C 90.000,E1 100.489} C_DIS
LIN {X 0.167,Y -554.645,Z 473.357,A 0.000,B 0.000,C 90.000,E1 100.310} C_DIS
LIN {X -0.018,Y -561.352,Z 473.356,A 0.000,B 0.000,C 90.000,E1 100.141} C_DIS
LIN {X 0.151,Y -564.800,Z 473.356,A 0.000,B 0.000,C 90.000,E1 100.018} C_DIS
LIN {X 0.102,Y -574.752,Z 473.354,A 0.000,B 0.000,C 90.000,E1 99.670} C_DIS
LIN {X -0.113,Y -581.354,Z 473.352,A 0.000,B 0.000,C 90.000,E1 99.434} C_DIS
LIN {X -0.142,Y -587.552,Z 473.351,A 0.000,B 0.000,C 90.000,E1 99.151} C_DIS
LIN {X 0.161,Y -593.915,Z 473.349,A 0.000,B 0.000,C 90.000,E1 98.803} C_DIS
LIN {X 0.209,Y -600.066,Z 473.347,A 0.000,B 0.000,C 90.000,E1 98.454} C_DIS
LIN {X -0.030,Y -605.870,Z 473.345,A 0.000,B 0.000,C 90.000,E1 98.106} C_DIS
LIN {X -0.035,Y -612.891,Z 473.342,A 0.000,B 0.000,C 90.000,E1 97.587} C_DIS
LIN {X 0.087,Y -618.155,Z 473.340,A 0.000,B 0.000,C 90.000,E1 97.125} C_DIS
LIN {X -0.094,Y -624.401,Z 473.336,A 0.000,B 0.000,C 90.000,E1 96.543} C_DIS
LIN {X -0.183,Y -630.774,Z 473.332,A 0.000,B 0.000,C 90.000,E1 95.796} C_DIS
LIN {X -0.054,Y -634.160,Z 473.329,A 0.000,B 0.000,C 90.000,E1 95.277} C_DIS
LIN {X 0.178,Y -637.392,Z 473.327,A 0.000,B 0.000,C 90.000,E1 94.759} C_DIS
LIN {X -0.209,Y -639.551,Z 473.324,A 0.000,B 0.000,C 90.000,E1 94.416} C_DIS
LIN {X -0.144,Y -642.796,Z 473.321,A 0.000,B 0.000,C 90.000,E1 93.784} C_DIS
LIN {X 0.023,Y -644.975,Z 473.318,A 0.000,B 0.000,C 90.000,E1 93.269} C_DIS
LIN {X -0.175,Y -645.954,Z 473.317,A 0.000,B 0.000,C 90.000,E1 93.037} C_DIS
LIN {X 0.015,Y -647.534,Z 473.314,A 0.000,B 0.000,C 90.000,E1 92.522} C_DIS
LIN {X 0.026,Y -649.454,Z 473.310,A 0.000,B 0.000,C 90.000,E1 91.776} C_DIS
LIN {X 0.244,Y -650.277,Z 473.307,A 0.000,B 0.000,C 90.000,E1 91.260} C_DIS
LIN {X -0.178,Y -650.836,Z 473.304,A 0.000,B 0.000,C 90.000,E1 90.802} C_DIS
LIN {X 0.263,Y -651.006,Z 473.303,A 0.000,B 0.000,C 90.000,E1 90.516} C_DIS
LIN {X -0.152,Y -651.103,Z 473.300,A 0.000,B 0.000,C 90.000,E1 90.057} C_DIS
LIN {X -0.124,Y -650.602,Z 473.296,A 0.000,B 0.000,C 90.000,E1 89.312} C_DIS
LIN {X 0.108,Y -649.906,Z 473.293,A 0.000,B 0.000,C 90.000,E1 88.797} C_DIS
LIN {X -0.315,Y -648.956,Z 473.291,A 0.000,B 0.000,C 90.000,E1 88.339} C_DIS
LIN {X -0.074,Y -647.664,Z 473.288,A 0.000,B 0.000,C 90.000,E1 87.822} C_DIS
LIN {X -0.087,Y -645.011,Z 473.284,A 0.000,B 0.000,C 90.000,E1 87.078} C_DIS
LIN {X 0.137,Y -643.018,Z 473.281,A 0.000,B 0.000,C 90.000,E1 86.560} C_DIS
LIN {X -0.214,Y -641.157,Z 473.279,A 0.000,B 0.000,C 90.000,E1 86.216} C_DIS
LIN {X 0.243,Y -636.118,Z 473.274,A 0.000,B 0.000,C 90.000,E1 85.298} C_DIS
LIN {X -0.224,Y -632.581,Z 473.271,A 0.000,B 0.000,C 90.000,E1 84.837} C_DIS
LIN {X -0.080,Y -628.814,Z 473.268,A 0.000,B 0.000,C 90.000,E1 84.318} C_DIS
LIN {X -0.110,Y -623.868,Z 473.265,A 0.000,B 0.000,C 90.000,E1 83.685} C_DIS
LIN {X -0.182,Y -618.016,Z 473.261,A 0.000,B 0.000,C 90.000,E1 83.053} C_DIS
LIN {X 0.227,Y -611.744,Z 473.258,A 0.000,B 0.000,C 90.000,E1 82.413} C_DIS
LIN {X 0.085,Y -606.301,Z 473.255,A 0.000,B 0.000,C 90.000,E1 81.951} C_DIS
LIN {X 0.154,Y -600.646,Z 473.253,A 0.000,B 0.000,C 90.000,E1 81.489} C_DIS
LIN {X 0.014,Y -595.095,Z 473.251,A 0.000,B 0.000,C 90.000,E1 81.084} C_DIS
LIN {X -0.078,Y -588.844,Z 473.248,A 0.000,B 0.000,C 90.000,E1 80.679} C_DIS
LIN {X -0.299,Y -582.441,Z 473.246,A 0.000,B 0.000,C 90.000,E1 80.330} C_DIS
LIN {X 0.088,Y -577.268,Z 473.245,A 0.000,B 0.000,C 90.000,E1 80.038} C_DIS
LIN {X 0.098,Y -571.776,Z 473.243,A 0.000,B 0.000,C 90.000,E1 79.803} C_DIS
LIN {X -0.143,Y -567.803,Z 473.243,A 0.000,B 0.000,C 90.000,E1 79.690} C_DIS
LIN {X -0.119,Y -563.855,Z 473.242,A 0.000,B 0.000,C 90.000,E1 79.567} C_DIS
LIN {X 0.176,Y -557.744,Z 473.241,A 0.000,B 0.000,C 90.000,E1 79.398} C_DIS
LIN {X -0.063,Y -551.909,Z 473.241,A 0.000,B 0.000,C 90.000,E1 79.342} C_DIS
LIN {X 0.098,Y -545.616,Z 473.241,A 0.000,B 0.000,C 90.000,E1 79.285} C_DIS
LIN {X 0.048,Y -482.264,Z 473.241,A 0.000,B 0.000,C 90.000,E1 79.285} C_DIS
LIN {X -0.103,Y -480.473,Z 473.227,A 0.000,B 0.000,C 90.000,E1 76.825} C_DIS
LIN {X -0.206,Y -474.232,Z 473.201,A 0.000,B 0.000,C 90.000,E1 72.181} C_DIS
LIN {X 0.212,Y -473.737,Z 473.199,A 0.000,B 0.000,C 90.000,E1 71.819} C_DIS
LIN {X -0.275,Y -466.180,Z 473.175,A 0.000,B 0.000,C 90.000,E1 67.486} C_DIS
LIN {X 0.277,Y -465.754,Z 473.173,A 0.000,B 0.000,C 90.000,E1 67.102} C_DIS
LIN {X 0.092,Y -463.649,Z 473.168,A 0.000,B 0.000,C 90.000,E1 66.177} C_DIS
LIN {X 0.073,Y -455.900,Z 473.145,A 0.000,B 0.000,C 90.000,E1 62.153} C_DIS
LIN {X 0.034,Y -455.916,Z 473.145,A 0.000,B 0.000,C 90.000,E1 62.153} C_DIS
LIN {X 0.048,Y -463.469,Z 473.139,A 0.000,B 0.000,C 90.000,E1 60.923} C_DIS
LIN {X 0.079,Y -468.096,Z 473.134,A 0.000,B 0.000,C 90.000,E1 60.127} C_DIS
LIN {X 0.159,Y -472.511,Z 473.130,A 0.000,B 0.000,C 90.000,E1 59.331} C_DIS
LIN {X 0.045,Y -477.284,Z 473.125,A 0.000,B 0.000,C 90.000,E1 58.408} C_DIS
LIN {X 0.031,Y -480.090,Z 473.121,A 0.000,B 0.000,C 90.000,E1 57.788} C_DIS
LIN {X 0.006,Y -481.960,Z 473.119,A 0.000,B 0.000,C 90.000,E1 57.327} C_DIS
LIN {X 0.025,Y -484.232,Z 473.115,A 0.000,B 0.000,C 90.000,E1 56.707} C_DIS
LIN {X 0.061,Y -486.151,Z 473.112,A 0.000,B 0.000,C 90.000,E1 56.087} C_DIS
LIN {X -0.059,Y -488.369,Z 473.107,A 0.000,B 0.000,C 90.000,E1 55.182} C_DIS
LIN {X 0.008,Y -489.631,Z 473.103,A 0.000,B 0.000,C 90.000,E1 54.562} C_DIS
LIN {X 0.213,Y -491.097,Z 473.098,A 0.000,B 0.000,C 90.000,E1 53.623} C_DIS
LIN {X 0.143,Y -492.083,Z 473.093,A 0.000,B 0.000,C 90.000,E1 52.718} C_DIS
LIN {X -0.009,Y -492.808,Z 473.088,A 0.000,B 0.000,C 90.000,E1 51.823} C_DIS
LIN {X 0.236,Y -493.305,Z 473.083,A 0.000,B 0.000,C 90.000,E1 50.884} C_DIS
LIN {X 0.102,Y -493.606,Z 473.078,A 0.000,B 0.000,C 90.000,E1 49.989} C_DIS
LIN {X -0.030,Y -493.786,Z 473.073,A 0.000,B 0.000,C 90.000,E1 49.094} C_DIS
LIN {X 0.166,Y -493.825,Z 473.068,A 0.000,B 0.000,C 90.000,E1 48.162} C_DIS
LIN {X -0.156,Y -493.649,Z 473.061,A 0.000,B 0.000,C 90.000,E1 46.986} C_DIS
LIN {X 0.040,Y -493.451,Z 473.056,A 0.000,B 0.000,C 90.000,E1 46.053} C_DIS
LIN {X 0.055,Y -493.030,Z 473.049,A 0.000,B 0.000,C 90.000,E1 44.838} C_DIS
LIN {X 0.062,Y -492.508,Z 473.042,A 0.000,B 0.000,C 90.000,E1 43.623} C_DIS
LIN {X 0.083,Y -491.810,Z 473.036,A 0.000,B 0.000,C 90.000,E1 42.405} C_DIS
LIN {X -0.107,Y -490.743,Z 473.027,A 0.000,B 0.000,C 90.000,E1 40.906} C_DIS
LIN {X -0.058,Y -489.406,Z 473.017,A 0.000,B 0.000,C 90.000,E1 39.072} C_DIS
LIN {X 0.129,Y -488.217,Z 473.009,A 0.000,B 0.000,C 90.000,E1 37.523} C_DIS
LIN {X -0.011,Y -486.937,Z 473.000,A 0.000,B 0.000,C 90.000,E1 36.011} C_DIS
LIN {X -0.065,Y -485.535,Z 472.992,A 0.000,B 0.000,C 90.000,E1 34.485} C_DIS
LIN {X -0.143,Y -483.951,Z 472.983,A 0.000,B 0.000,C 90.000,E1 32.959} C_DIS
LIN {X 0.111,Y -481.880,Z 472.973,A 0.000,B 0.000,C 90.000,E1 31.082} C_DIS
LIN {X -0.103,Y -480.447,Z 472.966,A 0.000,B 0.000,C 90.000,E1 29.873} C_DIS
LIN {X -0.179,Y -478.288,Z 472.956,A 0.000,B 0.000,C 90.000,E1 28.025} C_DIS
LIN {X -0.169,Y -475.565,Z 472.942,A 0.000,B 0.000,C 90.000,E1 25.540} C_DIS
LIN {X 0.116,Y -472.790,Z 472.924,A 0.000,B 0.000,C 90.000,E1 22.386} C_DIS
LIN {X 0.056,Y -470.925,Z 472.909,A 0.000,B 0.000,C 90.000,E1 19.577} C_DIS
LIN {X 0.074,Y -469.815,Z 472.898,A 0.000,B 0.000,C 90.000,E1 17.692} C_DIS
LIN {X -0.029,Y -468.908,Z 472.890,A 0.000,B 0.000,C 90.000,E1 16.134} C_DIS
LIN {X -0.090,Y -467.722,Z 472.877,A 0.000,B 0.000,C 90.000,E1 13.939} C_DIS
LIN {X 0.059,Y -466.878,Z 472.865,A 0.000,B 0.000,C 90.000,E1 11.715} C_DIS
LIN {X -0.161,Y -466.463,Z 472.855,A 0.000,B 0.000,C 90.000,E1 9.849} C_DIS
LIN {X -0.136,Y -466.234,Z 472.839,A 0.000,B 0.000,C 90.000,E1 7.004} C_DIS
LIN {X 0.143,Y -466.945,Z 472.820,A 0.000,B 0.000,C 90.000,E1 3.498} C_DIS
LIN {X 0.161,Y -468.663,Z 472.802,A 0.000,B 0.000,C 90.000,E1 0.344} C_DIS
LIN {X 0.232,Y -470.706,Z 472.788,A 0.000,B 0.000,C 90.000,E1 357.879} C_DIS
LIN {X -0.032,Y -474.070,Z 472.771,A 0.000,B 0.000,C 90.000,E1 354.780} C_DIS
LIN {X 0.247,Y -476.407,Z 472.761,A 0.000,B 0.000,C 90.000,E1 352.875} C_DIS
LIN {X -0.014,Y -480.807,Z 472.743,A 0.000,B 0.000,C 90.000,E1 349.803} C_DIS
LIN {X 0.030,Y -486.631,Z 472.725,A 0.000,B 0.000,C 90.000,E1 346.408} C_DIS
LIN {X -0.102,Y -491.052,Z 472.713,A 0.000,B 0.000,C 90.000,E1 344.283} C_DIS
LIN {X 0.258,Y -495.164,Z 472.703,A 0.000,B 0.000,C 90.000,E1 342.417} C_DIS
LIN {X 0.193,Y -498.715,Z 472.694,A 0.000,B 0.000,C 90.000,E1 340.913} C_DIS
LIN {X -0.141,Y -503.808,Z 472.682,A 0.000,B 0.000,C 90.000,E1 338.847} C_DIS
LIN {X -0.178,Y -507.448,Z 472.674,A 0.000,B 0.000,C 90.000,E1 337.358} C_DIS
LIN {X 0.169,Y -511.658,Z 472.664,A 0.000,B 0.000,C 90.000,E1 335.537} C_DIS
LIN {X -0.195,Y -516.523,Z 472.653,A 0.000,B 0.000,C 90.000,E1 333.512} C_DIS
LIN {X 0.109,Y -520.736,Z 472.643,A 0.000,B 0.000,C 90.000,E1 331.719} C_DIS
LIN {X -0.133,Y -527.059,Z 472.628,A 0.000,B 0.000,C 90.000,E1 329.125} C_DIS
LIN {X 0.010,Y -531.410,Z 472.619,A 0.000,B 0.000,C 90.000,E1 327.375} C_DIS
LIN {X -0.208,Y -536.548,Z 472.608,A 0.000,B 0.000,C 90.000,E1 325.388} C_DIS
LIN {X 0.294,Y -541.006,Z 472.598,A 0.000,B 0.000,C 90.000,E1 323.623} C_DIS
LIN {X -0.336,Y -544.817,Z 472.590,A 0.000,B 0.000,C 90.000,E1 322.271} C_DIS
LIN {X 0.242,Y -549.243,Z 472.581,A 0.000,B 0.000,C 90.000,E1 320.517} C_DIS
LIN {X 0.378,Y -552.250,Z 472.575,A 0.000,B 0.000,C 90.000,E1 319.380} C_DIS
LIN {X -0.138,Y -556.630,Z 472.565,A 0.000,B 0.000,C 90.000,E1 317.757} C_DIS
LIN {X -0.235,Y -560.277,Z 472.558,A 0.000,B 0.000,C 90.000,E1 316.377} C_DIS
LIN {X -0.291,Y -563.812,Z 472.550,A 0.000,B 0.000,C 90.000,E1 315.000} C_DIS
LIN {X -0.108,Y -568.770,Z 472.539,A 0.000,B 0.000,C 90.000,E1 313.056} C_DIS
LIN {X 0.310,Y -571.600,Z 472.533,A 0.000,B 0.000,C 90.000,E1 311.919} C_DIS
LIN {X -0.328,Y -575.014,Z 472.526,A 0.000,B 0.000,C 90.000,E1 310.620} C_DIS
LIN {X 0.049,Y -579.171,Z 472.516,A 0.000,B 0.000,C 90.000,E1 308.955} C_DIS
LIN {X 0.066,Y -582.611,Z 472.509,A 0.000,B 0.000,C 90.000,E1 307.604} C_DIS
LIN {X -0.314,Y -586.009,Z 472.502,A 0.000,B 0.000,C 90.000,E1 306.297} C_DIS
LIN {X -0.173,Y -589.375,Z 472.494,A 0.000,B 0.000,C 90.000,E1 304.945} C_DIS
LIN {X 0.386,Y -593.314,Z 472.485,A 0.000,B 0.000,C 90.000,E1 303.293} C_DIS
LIN {X 0.090,Y -595.826,Z 472.479,A 0.000,B 0.000,C 90.000,E1 302.260} C_DIS
LIN {X 0.020,Y -598.248,Z 472.473,A 0.000,B 0.000,C 90.000,E1 301.209} C_DIS
LIN {X 0.295,Y -600.478,Z 472.468,A 0.000,B 0.000,C 90.000,E1 300.129} C_DIS
LIN {X 0.296,Y -602.563,Z 472.462,A 0.000,B 0.000,C 90.000,E1 299.077} C_DIS
LIN {X 0.264,Y -605.004,Z 472.454,A 0.000,B 0.000,C 90.000,E1 297.769} C_DIS
LIN {X 0.042,Y -606.872,Z 472.449,A 0.000,B 0.000,C 90.000,E1 296.744} C_DIS
LIN {X -0.202,Y -608.966,Z 472.441,A 0.000,B 0.000,C 90.000,E1 295.463} C_DIS
LIN {X 0.177,Y -610.390,Z 472.436,A 0.000,B 0.000,C 90.000,E1 294.387} C_DIS
LIN {X 0.287,Y -612.015,Z 472.428,A 0.000,B 0.000,C 90.000,E1 293.078} C_DIS
LIN {X -0.105,Y -613.306,Z 472.423,A 0.000,B 0.000,C 90.000,E1 292.078} C_DIS
LIN {X -0.138,Y -614.479,Z 472.417,A 0.000,B 0.000,C 90.000,E1 291.046} C_DIS
LIN {X -0.184,Y -615.825,Z 472.410,A 0.000,B 0.000,C 90.000,E1 289.758} C_DIS
LIN {X 0.125,Y -617.311,Z 472.401,A 0.000,B 0.000,C 90.000,E1 288.181} C_DIS
LIN {X 0.196,Y -617.927,Z 472.397,A 0.000,B 0.000,C 90.000,E1 287.402} C_DIS
LIN {X -0.087,Y -618.449,Z 472.394,A 0.000,B 0.000,C 90.000,E1 286.913} C_DIS
LIN {X -0.317,Y -619.840,Z 472.384,A 0.000,B 0.000,C 90.000,E1 285.134} C_DIS
LIN {X -0.070,Y -620.584,Z 472.377,A 0.000,B 0.000,C 90.000,E1 283.828} C_DIS
LIN {X 0.038,Y -621.191,Z 472.370,A 0.000,B 0.000,C 90.000,E1 282.535} C_DIS
LIN {X 0.153,Y -621.610,Z 472.363,A 0.000,B 0.000,C 90.000,E1 281.243} C_DIS
LIN {X 0.150,Y -621.812,Z 472.355,A 0.000,B 0.000,C 90.000,E1 279.962} C_DIS
LIN {X 0.146,Y -621.699,Z 472.348,A 0.000,B 0.000,C 90.000,E1 278.681} C_DIS
LIN {X 0.042,Y -621.383,Z 472.341,A 0.000,B 0.000,C 90.000,E1 277.409} C_DIS
LIN {X 0.171,Y -620.846,Z 472.336,A 0.000,B 0.000,C 90.000,E1 276.372} C_DIS
LIN {X 0.293,Y -620.216,Z 472.330,A 0.000,B 0.000,C 90.000,E1 275.334} C_DIS
LIN {X 0.046,Y -618.975,Z 472.323,A 0.000,B 0.000,C 90.000,E1 274.073} C_DIS
LIN {X -0.176,Y -617.428,Z 472.316,A 0.000,B 0.000,C 90.000,E1 272.808} C_DIS
LIN {X -0.155,Y -615.941,Z 472.310,A 0.000,B 0.000,C 90.000,E1 271.776} C_DIS
LIN {X 0.141,Y -614.697,Z 472.306,A 0.000,B 0.000,C 90.000,E1 270.974} C_DIS
LIN {X -0.206,Y -612.529,Z 472.298,A 0.000,B 0.000,C 90.000,E1 269.714} C_DIS
LIN {X -0.290,Y -609.644,Z 472.290,A 0.000,B 0.000,C 90.000,E1 268.165} C_DIS
LIN {X -0.091,Y -607.083,Z 472.282,A 0.000,B 0.000,C 90.000,E1 266.846} C_DIS
LIN {X 0.055,Y -604.308,Z 472.275,A 0.000,B 0.000,C 90.000,E1 265.527} C_DIS
LIN {X -0.049,Y -601.993,Z 472.269,A 0.000,B 0.000,C 90.000,E1 264.489} C_DIS
LIN {X -0.037,Y -597.759,Z 472.259,A 0.000,B 0.000,C 90.000,E1 262.648} C_DIS
LIN {X 0.019,Y -593.371,Z 472.249,A 0.000,B 0.000,C 90.000,E1 260.792} C_DIS
LIN {X 0.120,Y -590.072,Z 472.242,A 0.000,B 0.000,C 90.000,E1 259.454} C_DIS
LIN {X 0.156,Y -586.644,Z 472.234,A 0.000,B 0.000,C 90.000,E1 258.117} C_DIS
LIN {X 0.048,Y -582.415,Z 472.225,A 0.000,B 0.000,C 90.000,E1 256.520} C_DIS
LIN {X 0.063,Y -578.822,Z 472.218,A 0.000,B 0.000,C 90.000,E1 255.172} C_DIS
LIN {X 0.307,Y -575.148,Z 472.210,A 0.000,B 0.000,C 90.000,E1 253.795} C_DIS
LIN {X 0.124,Y -570.583,Z 472.201,A 0.000,B 0.000,C 90.000,E1 252.181} C_DIS
LIN {X -0.319,Y -566.583,Z 472.194,A 0.000,B 0.000,C 90.000,E1 250.859} C_DIS
LIN {X -0.325,Y -561.577,Z 472.184,A 0.000,B 0.000,C 90.000,E1 249.209} C_DIS
LIN {X -0.017,Y -557.207,Z 472.177,A 0.000,B 0.000,C 90.000,E1 247.794} C_DIS
LIN {X -0.087,Y -552.551,Z 472.169,A 0.000,B 0.000,C 90.000,E1 246.410} C_DIS
LIN {X 0.007,Y -548.730,Z 472.163,A 0.000,B 0.000,C 90.000,E1 245.281} C_DIS
LIN {X 0.028,Y -542.816,Z 472.153,A 0.000,B 0.000,C 90.000,E1 243.589} C_DIS
LIN {X 0.184,Y -537.864,Z 472.145,A 0.000,B 0.000,C 90.000,E1 242.153} C_DIS
LIN {X 0.259,Y -532.959,Z 472.138,A 0.000,B 0.000,C 90.000,E1 240.717} C_DIS
LIN {X -0.110,Y -526.007,Z 472.126,A 0.000,B 0.000,C 90.000,E1 238.742} C_DIS
LIN {X 0.280,Y -521.150,Z 472.118,A 0.000,B 0.000,C 90.000,E1 237.248} C_DIS
LIN {X 0.079,Y -515.247,Z 472.109,A 0.000,B 0.000,C 90.000,E1 235.515} C_DIS
LIN {X -0.086,Y -511.112,Z 472.102,A 0.000,B 0.000,C 90.000,E1 234.356} C_DIS
LIN {X -0.272,Y -499.220,Z 472.082,A 0.000,B 0.000,C 90.000,E1 230.803} C_DIS
LIN {X 0.113,Y -492.968,Z 472.070,A 0.000,B 0.000,C 90.000,E1 228.647} C_DIS
LIN {X 0.068,Y -486.010,Z 472.057,A 0.000,B 0.000,C 90.000,E1 226.215} C_DIS
LIN {X 0.236,Y -480.941,Z 472.047,A 0.000,B 0.000,C 90.000,E1 224.352} C_DIS
LIN {X 0.063,Y -475.294,Z 472.035,A 0.000,B 0.000,C 90.000,E1 222.204} C_DIS
LIN {X -0.101,Y -469.280,Z 472.021,A 0.000,B 0.000,C 90.000,E1 219.725} C_DIS
LIN {X 0.282,Y -463.654,Z 472.007,A 0.000,B 0.000,C 90.000,E1 217.156} C_DIS
LIN {X -0.080,Y -459.057,Z 471.994,A 0.000,B 0.000,C 90.000,E1 214.978} C_DIS
LIN {X -0.183,Y -454.634,Z 471.982,A 0.000,B 0.000,C 90.000,E1 212.752} C_DIS
LIN {X 0.017,Y -450.993,Z 471.971,A 0.000,B 0.000,C 90.000,E1 210.797} C_DIS
LIN {X -0.179,Y -446.181,Z 471.957,A 0.000,B 0.000,C 90.000,E1 208.231} C_DIS
LIN {X 0.156,Y -442.521,Z 471.946,A 0.000,B 0.000,C 90.000,E1 206.232} C_DIS
LIN {X -0.224,Y -439.457,Z 471.937,A 0.000,B 0.000,C 90.000,E1 204.643} C_DIS
LIN {X 0.033,Y -434.504,Z 471.922,A 0.000,B 0.000,C 90.000,E1 201.972} C_DIS
LIN {X 0.156,Y -430.398,Z 471.909,A 0.000,B 0.000,C 90.000,E1 199.631} C_DIS
LIN {X -0.134,Y -426.549,Z 471.896,A 0.000,B 0.000,C 90.000,E1 197.330} C_DIS
LIN {X 0.039,Y -423.056,Z 471.883,A 0.000,B 0.000,C 90.000,E1 194.954} C_DIS
LIN {X 0.013,Y -419.876,Z 471.870,A 0.000,B 0.000,C 90.000,E1 192.591} C_DIS
LIN {X -0.169,Y -416.177,Z 471.853,A 0.000,B 0.000,C 90.000,E1 189.557} C_DIS
LIN {X 0.157,Y -413.137,Z 471.838,A 0.000,B 0.000,C 90.000,E1 186.777} C_DIS
LIN {X -0.151,Y -410.751,Z 471.824,A 0.000,B 0.000,C 90.000,E1 184.416} C_DIS
LIN {X -0.159,Y -408.927,Z 471.813,A 0.000,B 0.000,C 90.000,E1 182.350} C_DIS
LIN {X 0.165,Y -407.180,Z 471.800,A 0.000,B 0.000,C 90.000,E1 179.885} C_DIS
LIN {X -0.023,Y -405.449,Z 471.780,A 0.000,B 0.000,C 90.000,E1 176.445} C_DIS
LIN {X -0.158,Y -404.655,Z 471.763,A 0.000,B 0.000,C 90.000,E1 173.337} C_DIS
LIN {X -0.163,Y -404.730,Z 471.746,A 0.000,B 0.000,C 90.000,E1 170.208} C_DIS
LIN {X -0.130,Y -405.221,Z 471.734,A 0.000,B 0.000,C 90.000,E1 168.117} C_DIS
LIN {X 0.170,Y -406.245,Z 471.720,A 0.000,B 0.000,C 90.000,E1 165.644} C_DIS
LIN {X -0.073,Y -407.765,Z 471.705,A 0.000,B 0.000,C 90.000,E1 162.906} C_DIS
LIN {X -0.148,Y -409.630,Z 471.692,A 0.000,B 0.000,C 90.000,E1 160.496} C_DIS
LIN {X 0.101,Y -411.828,Z 471.678,A 0.000,B 0.000,C 90.000,E1 158.050} C_DIS
LIN {X -0.032,Y -414.350,Z 471.665,A 0.000,B 0.000,C 90.000,E1 155.665} C_DIS
LIN {X 0.084,Y -415.881,Z 471.657,A 0.000,B 0.000,C 90.000,E1 154.280} C_DIS
LIN {X 0.058,Y -418.721,Z 471.644,A 0.000,B 0.000,C 90.000,E1 151.897} C_DIS
LIN {X 0.050,Y -420.343,Z 471.636,A 0.000,B 0.000,C 90.000,E1 150.539} C_DIS
LIN {X -0.094,Y -422.010,Z 471.629,A 0.000,B 0.000,C 90.000,E1 149.203} C_DIS
LIN {X -0.032,Y -424.455,Z 471.618,A 0.000,B 0.000,C 90.000,E1 147.168} C_DIS
LIN {X -0.269,Y -427.001,Z 471.606,A 0.000,B 0.000,C 90.000,E1 145.182} C_DIS
LIN {X 0.038,Y -429.670,Z 471.595,A 0.000,B 0.000,C 90.000,E1 143.130} C_DIS
LIN {X 0.059,Y -432.388,Z 471.584,A 0.000,B 0.000,C 90.000,E1 141.126} C_DIS
LIN {X 0.082,Y -434.685,Z 471.575,A 0.000,B 0.000,C 90.000,E1 139.461} C_DIS
LIN {X 0.154,Y -436.849,Z 471.566,A 0.000,B 0.000,C 90.000,E1 137.796} C_DIS
LIN {X -0.036,Y -438.541,Z 471.558,A 0.000,B 0.000,C 90.000,E1 136.500} C_DIS
LIN {X 0.123,Y -439.828,Z 471.551,A 0.000,B 0.000,C 90.000,E1 135.162} C_DIS
LIN {X -0.016,Y -440.866,Z 471.544,A 0.000,B 0.000,C 90.000,E1 133.866} C_DIS
LIN {X 0.177,Y -441.563,Z 471.536,A 0.000,B 0.000,C 90.000,E1 132.528} C_DIS
LIN {X -0.217,Y -441.826,Z 471.531,A 0.000,B 0.000,C 90.000,E1 131.595} C_DIS
LIN {X -0.276,Y -441.719,Z 471.526,A 0.000,B 0.000,C 90.000,E1 130.620} C_DIS
LIN {X 0.288,Y -441.178,Z 471.520,A 0.000,B 0.000,C 90.000,E1 129.564} C_DIS
LIN {X -0.055,Y -440.397,Z 471.515,A 0.000,B 0.000,C 90.000,E1 128.624} C_DIS
LIN {X -0.133,Y -439.317,Z 471.509,A 0.000,B 0.000,C 90.000,E1 127.649} C_DIS
LIN {X -0.145,Y -437.993,Z 471.504,A 0.000,B 0.000,C 90.000,E1 126.664} C_DIS
LIN {X 0.108,Y -435.842,Z 471.496,A 0.000,B 0.000,C 90.000,E1 125.311} C_DIS
LIN {X 0.088,Y -432.737,Z 471.487,A 0.000,B 0.000,C 90.000,E1 123.658} C_DIS
LIN {X 0.005,Y -429.147,Z 471.478,A 0.000,B 0.000,C 90.000,E1 122.005} C_DIS
LIN {X -0.228,Y -427.653,Z 471.474,A 0.000,B 0.000,C 90.000,E1 121.337} C_DIS
LIN {X -0.267,Y -427.663,Z 471.474,A 0.000,B 0.000,C 90.000,E1 121.337} C_DIS
LIN {X -0.007,Y -430.626,Z 471.469,A 0.000,B 0.000,C 90.000,E1 120.335} C_DIS
LIN {X -0.013,Y -441.531,Z 471.445,A 0.000,B 0.000,C 90.000,E1 116.027} C_DIS
LIN {X 0.114,Y -444.447,Z 471.439,A 0.000,B 0.000,C 90.000,E1 115.027} C_DIS
LIN {X 0.012,Y -445.919,Z 471.436,A 0.000,B 0.000,C 90.000,E1 114.387} C_DIS
LIN {X 0.150,Y -455.325,Z 471.414,A 0.000,B 0.000,C 90.000,E1 110.482} C_DIS
LIN {X -0.055,Y -457.125,Z 471.410,A 0.000,B 0.000,C 90.000,E1 109.866} C_DIS
LIN {X -0.207,Y -466.525,Z 471.386,A 0.000,B 0.000,C 90.000,E1 105.426} C_DIS
LIN {X -0.031,Y -467.986,Z 471.382,A 0.000,B 0.000,C 90.000,E1 104.773} C_DIS
LIN {X -0.094,Y -475.520,Z 471.358,A 0.000,B 0.000,C 90.000,E1 100.423} C_DIS
LIN {X -0.149,Y -516.014,Z 471.358,A 0.000,B 0.000,C 90.000,E1 100.423} C_DIS
LIN {X 0.266,Y -518.847,Z 471.358,A 0.000,B 0.000,C 90.000,E1 100.366} C_DIS
LIN {X 0.235,Y -524.559,Z 471.358,A 0.000,B 0.000,C 90.000,E1 100.366} C_DIS
LIN {X 0.246,Y -532.030,Z 471.357,A 0.000,B 0.000,C 90.000,E1 100.310} C_DIS
LIN {X 0.217,Y -538.247,Z 471.357,A 0.000,B 0.000,C 90.000,E1 100.254} C_DIS
LIN {X 0.201,Y -548.123,Z 471.356,A 0.000,B 0.000,C 90.000,E1 100.074} C_DIS
LIN {X -0.070,Y -554.505,Z 471.355,A 0.000,B 0.000,C 90.000,E1 99.962} C_DIS
LIN {X -0.122,Y -561.366,Z 471.354,A 0.000,B 0.000,C 90.000,E1 99.792} C_DIS
LIN {X 0.160,Y -564.641,Z 471.354,A 0.000,B 0.000,C 90.000,E1 99.670} C_DIS
LIN {X 0.265,Y -574.481,Z 471.352,A 0.000,B 0.000,C 90.000,E1 99.321} C_DIS
LIN {X 0.078,Y -581.195,Z 471.351,A 0.000,B 0.000,C 90.000,E1 99.095} C_DIS
LIN {X 0.233,Y -587.564,Z 471.349,A 0.000,B 0.000,C 90.000,E1 98.803} C_DIS
LIN {X 0.110,Y -596.972,Z 471.346,A 0.000,B 0.000,C 90.000,E1 98.341} C_DIS
LIN {X 0.221,Y -599.977,Z 471.346,A 0.000,B 0.000,C 90.000,E1 98.163} C_DIS
LIN {X -0.015,Y -605.878,Z 471.343,A 0.000,B 0.000,C 90.000,E1 97.814} C_DIS
LIN {X 0.045,Y -611.545,Z 471.341,A 0.000,B 0.000,C 90.000,E1 97.409} C_DIS
LIN {X 0.265,Y -618.203,Z 471.338,A 0.000,B 0.000,C 90.000,E1 96.834} C_DIS
LIN {X -0.026,Y -624.458,Z 471.335,A 0.000,B 0.000,C 90.000,E1 96.258} C_DIS
LIN {X -0.009,Y -629.874,Z 471.331,A 0.000,B 0.000,C 90.000,E1 95.625} C_DIS
LIN {X -0.235,Y -631.716,Z 471.330,A 0.000,B 0.000,C 90.000,E1 95.391} C_DIS
LIN {X 0.264,Y -636.647,Z 471.326,A 0.000,B 0.000,C 90.000,E1 94.588} C_DIS
LIN {X -0.125,Y -638.832,Z 471.324,A 0.000,B 0.000,C 90.000,E1 94.245} C_DIS
LIN {X -0.065,Y -642.083,Z 471.320,A 0.000,B 0.000,C 90.000,E1 93.612} C_DIS
LIN {X 0.017,Y -644.697,Z 471.317,A 0.000,B 0.000,C 90.000,E1 92.980} C_DIS
LIN {X 0.199,Y -646.269,Z 471.314,A 0.000,B 0.000,C 90.000,E1 92.465} C_DIS
LIN {X 0.196,Y -648.153,Z 471.310,A 0.000,B 0.000,C 90.000,E1 91.718} C_DIS
LIN {X -0.241,Y -648.980,Z 471.307,A 0.000,B 0.000,C 90.000,E1 91.260} C_DIS
LIN {X -0.023,Y -649.512,Z 471.304,A 0.000,B 0.000,C 90.000,E1 90.745} C_DIS
LIN {X 0.201,Y -649.658,Z 471.301,A 0.000,B 0.000,C 90.000,E1 90.229} C_DIS
LIN {X -0.010,Y -649.667,Z 471.300,A 0.000,B 0.000,C 90.000,E1 90.000} C_DIS
LIN {X 0.216,Y -649.352,Z 471.297,A 0.000,B 0.000,C 90.000,E1 89.484} C_DIS
LIN {X -0.208,Y -648.721,Z 471.295,A 0.000,B 0.000,C 90.000,E1 89.026} C_DIS
LIN {X 0.009,Y -647.774,Z 471.292,A 0.000,B 0.000,C 90.000,E1 88.511} C_DIS
LIN {X 0.242,Y -646.489,Z 471.289,A 0.000,B 0.000,C 90.000,E1 87.993} C_DIS
LIN {X 0.022,Y -645.711,Z 471.288,A 0.000,B 0.000,C 90.000,E1 87.764} C_DIS
LIN {X -0.209,Y -641.872,Z 471.282,A 0.000,B 0.000,C 90.000,E1 86.788} C_DIS
LIN {X 0.197,Y -640.737,Z 471.281,A 0.000,B 0.000,C 90.000,E1 86.502} C_DIS
LIN {X -0.112,Y -634.982,Z 471.275,A 0.000,B 0.000,C 90.000,E1 85.527} C_DIS
LIN {X -0.226,Y -629.669,Z 471.271,A 0.000,B 0.000,C 90.000,E1 84.780} C_DIS
LIN {X 0.226,Y -623.591,Z 471.267,A 0.000,B 0.000,C 90.000,E1 83.976} C_DIS
LIN {X 0.216,Y -617.866,Z 471.263,A 0.000,B 0.000,C 90.000,E1 83.337} C_DIS
LIN {X -0.250,Y -611.363,Z 471.260,A 0.000,B 0.000,C 90.000,E1 82.761} C_DIS
LIN {X 0.191,Y -605.808,Z 471.257,A 0.000,B 0.000,C 90.000,E1 82.243} C_DIS
LIN {X 0.276,Y -599.973,Z 471.255,A 0.000,B 0.000,C 90.000,E1 81.781} C_DIS
LIN {X -0.293,Y -598.192,Z 471.254,A 0.000,B 0.000,C 90.000,E1 81.724} C_DIS
LIN {X -0.206,Y -595.353,Z 471.253,A 0.000,B 0.000,C 90.000,E1 81.489} C_DIS
LIN {X -0.067,Y -592.125,Z 471.251,A 0.000,B 0.000,C 90.000,E1 81.254} C_DIS
LIN {X 0.167,Y -588.894,Z 471.250,A 0.000,B 0.000,C 90.000,E1 81.027} C_DIS
LIN {X 0.084,Y -582.747,Z 471.248,A 0.000,B 0.000,C 90.000,E1 80.679} C_DIS
LIN {X -0.045,Y -577.331,Z 471.247,A 0.000,B 0.000,C 90.000,E1 80.443} C_DIS
LIN {X 0.169,Y -573.450,Z 471.246,A 0.000,B 0.000,C 90.000,E1 80.274} C_DIS
LIN {X 0.177,Y -570.583,Z 471.245,A 0.000,B 0.000,C 90.000,E1 80.151} C_DIS
LIN {X 0.002,Y -566.351,Z 471.245,A 0.000,B 0.000,C 90.000,E1 80.038} C_DIS
LIN {X 0.137,Y -562.815,Z 471.244,A 0.000,B 0.000,C 90.000,E1 79.926} C_DIS
LIN {X -0.187,Y -558.074,Z 471.244,A 0.000,B 0.000,C 90.000,E1 79.859} C_DIS
LIN {X 0.156,Y -551.556,Z 471.243,A 0.000,B 0.000,C 90.000,E1 79.746} C_DIS
LIN {X -0.060,Y -545.774,Z 471.243,A 0.000,B 0.000,C 90.000,E1 79.746} C_DIS
LIN {X -0.101,Y -482.676,Z 471.243,A 0.000,B 0.000,C 90.000,E1 79.746} C_DIS
LIN {X 0.032,Y -480.584,Z 471.228,A 0.000,B 0.000,C 90.000,E1 76.937} C_DIS
LIN {X -0.255,Y -479.663,Z 471.224,A 0.000,B 0.000,C 90.000,E1 76.353} C_DIS
LIN {X -0.221,Y -474.002,Z 471.200,A 0.000,B 0.000,C 90.000,E1 72.000} C_DIS
LIN {X -0.077,Y -466.361,Z 471.176,A 0.000,B 0.000,C 90.000,E1 67.592} C_DIS
LIN {X 0.239,Y -465.413,Z 471.172,A 0.000,B 0.000,C 90.000,E1 66.922} C_DIS
LIN {X -0.002,Y -456.991,Z 471.149,A 0.000,B 0.000,C 90.000,E1 62.820} C_DIS
LIN {X -0.116,Y -456.278,Z 471.147,A 0.000,B 0.000,C 90.000,E1 62.410} C_DIS
LIN {X -0.156,Y -456.272,Z 471.147,A 0.000,B 0.000,C 90.000,E1 62.410} C_DIS
LIN {X 0.096,Y -464.536,Z 471.139,A 0.000,B 0.000,C 90.000,E1 61.051} C_DIS
LIN {X 0.138,Y -469.219,Z 471.135,A 0.000,B 0.000,C 90.000,E1 60.255} C_DIS
LIN {X -0.010,Y -473.704,Z 471.131,A 0.000,B 0.000,C 90.000,E1 59.488} C_DIS
LIN {X -0.058,Y -476.959,Z 471.127,A 0.000,B 0.000,C 90.000,E1 58.869} C_DIS
LIN {X -0.077,Y -479.986,Z 471.124,A 0.000,B 0.000,C 90.000,E1 58.250} C_DIS
LIN {X 0.081,Y -482.672,Z 471.120,A 0.000,B 0.000,C 90.000,E1 57.612} C_DIS
LIN {X 0.144,Y -485.534,Z 471.116,A 0.000,B 0.000,C 90.000,E1 56.834} C_DIS
LIN {X 0.192,Y -487.524,Z 471.112,A 0.000,B 0.000,C 90.000,E1 56.215} C_DIS
LIN {X 0.090,Y -489.755,Z 471.107,A 0.000,B 0.000,C 90.000,E1 55.308} C_DIS
LIN {X 0.170,Y -491.028,Z 471.104,A 0.000,B 0.000,C 90.000,E1 54.689} C_DIS
LIN {X 0.103,Y -492.503,Z 471.099,A 0.000,B 0.000,C 90.000,E1 53.783} C_DIS
LIN {X -0.049,Y -493.481,Z 471.094,A 0.000,B 0.000,C 90.000,E1 52.889} C_DIS
LIN {X -0.095,Y -494.195,Z 471.089,A 0.000,B 0.000,C 90.000,E1 51.984} C_DIS
LIN {X -0.221,Y -494.681,Z 471.084,A 0.000,B 0.000,C 90.000,E1 51.090} C_DIS
LIN {X 0.043,Y -494.967,Z 471.079,A 0.000,B 0.000,C 90.000,E1 50.150} C_DIS
LIN {X -0.075,Y -495.111,Z 471.074,A 0.000,B 0.000,C 90.000,E1 49.256} C_DIS
LIN {X -0.017,Y -495.051,Z 471.067,A 0.000,B 0.000,C 90.000,E1 48.038} C_DIS
LIN {X -0.171,Y -494.888,Z 471.062,A 0.000,B 0.000,C 90.000,E1 47.148} C_DIS
LIN {X 0.221,Y -494.532,Z 471.055,A 0.000,B 0.000,C 90.000,E1 45.891} C_DIS
LIN {X -0.265,Y -493.947,Z 471.047,A 0.000,B 0.000,C 90.000,E1 44.433} C_DIS
LIN {X 0.113,Y -493.321,Z 471.040,A 0.000,B 0.000,C 90.000,E1 43.176} C_DIS
LIN {X -0.214,Y -492.496,Z 471.033,A 0.000,B 0.000,C 90.000,E1 42.000} C_DIS
LIN {X -0.182,Y -491.181,Z 471.023,A 0.000,B 0.000,C 90.000,E1 40.172} C_DIS
LIN {X 0.040,Y -490.000,Z 471.015,A 0.000,B 0.000,C 90.000,E1 38.624} C_DIS
LIN {X 0.098,Y -489.042,Z 471.008,A 0.000,B 0.000,C 90.000,E1 37.397} C_DIS
LIN {X 0.141,Y -488.014,Z 471.001,A 0.000,B 0.000,C 90.000,E1 36.171} C_DIS
LIN {X -0.012,Y -486.585,Z 470.993,A 0.000,B 0.000,C 90.000,E1 34.659} C_DIS
LIN {X 0.060,Y -485.001,Z 470.984,A 0.000,B 0.000,C 90.000,E1 33.118} C_DIS
LIN {X 0.185,Y -482.929,Z 470.974,A 0.000,B 0.000,C 90.000,E1 31.258} C_DIS
LIN {X -0.021,Y -481.485,Z 470.967,A 0.000,B 0.000,C 90.000,E1 30.050} C_DIS
LIN {X 0.113,Y -479.296,Z 470.957,A 0.000,B 0.000,C 90.000,E1 28.180} C_DIS
LIN {X -0.029,Y -476.814,Z 470.945,A 0.000,B 0.000,C 90.000,E1 26.027} C_DIS
LIN {X 0.023,Y -474.949,Z 470.934,A 0.000,B 0.000,C 90.000,E1 24.155} C_DIS
LIN {X -0.013,Y -472.943,Z 470.920,A 0.000,B 0.000,C 90.000,E1 21.663} C_DIS
LIN {X 0.222,Y -471.758,Z 470.910,A 0.000,B 0.000,C 90.000,E1 19.758} C_DIS
LIN {X 0.069,Y -470.450,Z 470.898,A 0.000,B 0.000,C 90.000,E1 17.583} C_DIS
LIN {X -0.076,Y -469.317,Z 470.887,A 0.000,B 0.000,C 90.000,E1 15.717} C_DIS
LIN {X 0.139,Y -468.044,Z 470.873,A 0.000,B 0.000,C 90.000,E1 13.175} C_DIS
LIN {X 0.189,Y -467.090,Z 470.856,A 0.000,B 0.000,C 90.000,E1 10.018} C_DIS
LIN {X 0.166,Y -466.761,Z 470.840,A 0.000,B 0.000,C 90.000,E1 7.182} C_DIS
LIN {X 0.048,Y -467.342,Z 470.821,A 0.000,B 0.000,C 90.000,E1 3.726} C_DIS
LIN {X 0.078,Y -468.969,Z 470.803,A 0.000,B 0.000,C 90.000,E1 0.573} C_DIS
LIN {X -0.229,Y -471.110,Z 470.788,A 0.000,B 0.000,C 90.000,E1 357.936} C_DIS
LIN {X 0.216,Y -474.127,Z 470.773,A 0.000,B 0.000,C 90.000,E1 355.065} C_DIS
LIN {X 0.059,Y -477.214,Z 470.759,A 0.000,B 0.000,C 90.000,E1 352.591} C_DIS
LIN {X -0.104,Y -481.718,Z 470.742,A 0.000,B 0.000,C 90.000,E1 349.511} C_DIS
LIN {X 0.204,Y -489.575,Z 470.718,A 0.000,B 0.000,C 90.000,E1 345.172} C_DIS
LIN {X -0.162,Y -494.920,Z 470.704,A 0.000,B 0.000,C 90.000,E1 342.779} C_DIS
LIN {X -0.234,Y -498.488,Z 470.696,A 0.000,B 0.000,C 90.000,E1 341.275} C_DIS
LIN {X -0.002,Y -502.842,Z 470.686,A 0.000,B 0.000,C 90.000,E1 339.444} C_DIS
LIN {X 0.143,Y -505.814,Z 470.679,A 0.000,B 0.000,C 90.000,E1 338.230} C_DIS
LIN {X 0.146,Y -509.436,Z 470.671,A 0.000,B 0.000,C 90.000,E1 336.741} C_DIS
LIN {X 0.311,Y -512.301,Z 470.664,A 0.000,B 0.000,C 90.000,E1 335.537} C_DIS
LIN {X -0.158,Y -516.481,Z 470.655,A 0.000,B 0.000,C 90.000,E1 333.819} C_DIS
LIN {X 0.115,Y -519.326,Z 470.648,A 0.000,B 0.000,C 90.000,E1 332.615} C_DIS
LIN {X -0.117,Y -522.821,Z 470.640,A 0.000,B 0.000,C 90.000,E1 331.179} C_DIS
LIN {X 0.070,Y -527.844,Z 470.629,A 0.000,B 0.000,C 90.000,E1 329.125} C_DIS
LIN {X 0.234,Y -532.240,Z 470.619,A 0.000,B 0.000,C 90.000,E1 327.375} C_DIS
LIN {X 0.038,Y -537.398,Z 470.608,A 0.000,B 0.000,C 90.000,E1 325.388} C_DIS
LIN {X -0.195,Y -541.874,Z 470.598,A 0.000,B 0.000,C 90.000,E1 323.703} C_DIS
LIN {X -0.051,Y -545.711,Z 470.590,A 0.000,B 0.000,C 90.000,E1 322.271} C_DIS
LIN {X -0.272,Y -549.455,Z 470.583,A 0.000,B 0.000,C 90.000,E1 320.884} C_DIS
LIN {X -0.078,Y -553.210,Z 470.575,A 0.000,B 0.000,C 90.000,E1 319.461} C_DIS
LIN {X 0.278,Y -558.411,Z 470.564,A 0.000,B 0.000,C 90.000,E1 317.472} C_DIS
LIN {X 0.268,Y -562.766,Z 470.555,A 0.000,B 0.000,C 90.000,E1 315.810} C_DIS
LIN {X -0.223,Y -565.643,Z 470.549,A 0.000,B 0.000,C 90.000,E1 314.757} C_DIS
LIN {X 0.004,Y -570.677,Z 470.538,A 0.000,B 0.000,C 90.000,E1 312.813} C_DIS
LIN {X -0.359,Y -573.492,Z 470.532,A 0.000,B 0.000,C 90.000,E1 311.757} C_DIS
LIN {X -0.010,Y -577.655,Z 470.523,A 0.000,B 0.000,C 90.000,E1 310.092} C_DIS
LIN {X -0.110,Y -581.164,Z 470.515,A 0.000,B 0.000,C 90.000,E1 308.749} C_DIS
LIN {X -0.334,Y -585.347,Z 470.506,A 0.000,B 0.000,C 90.000,E1 307.156} C_DIS
LIN {X -0.200,Y -588.735,Z 470.499,A 0.000,B 0.000,C 90.000,E1 305.804} C_DIS
LIN {X -0.013,Y -592.093,Z 470.491,A 0.000,B 0.000,C 90.000,E1 304.452} C_DIS
LIN {X 0.169,Y -594.736,Z 470.486,A 0.000,B 0.000,C 90.000,E1 303.372} C_DIS
LIN {X -0.104,Y -597.244,Z 470.480,A 0.000,B 0.000,C 90.000,E1 302.339} C_DIS
LIN {X 0.072,Y -600.244,Z 470.472,A 0.000,B 0.000,C 90.000,E1 301.003} C_DIS
LIN {X 0.303,Y -603.001,Z 470.465,A 0.000,B 0.000,C 90.000,E1 299.667} C_DIS
LIN {X 0.280,Y -605.491,Z 470.458,A 0.000,B 0.000,C 90.000,E1 298.359} C_DIS
LIN {X -0.031,Y -608.360,Z 470.449,A 0.000,B 0.000,C 90.000,E1 296.821} C_DIS
LIN {X -0.203,Y -610.102,Z 470.443,A 0.000,B 0.000,C 90.000,E1 295.796} C_DIS
LIN {X 0.198,Y -611.656,Z 470.437,A 0.000,B 0.000,C 90.000,E1 294.719} C_DIS
LIN {X -0.224,Y -613.369,Z 470.430,A 0.000,B 0.000,C 90.000,E1 293.462} C_DIS
LIN {X 0.210,Y -614.708,Z 470.425,A 0.000,B 0.000,C 90.000,E1 292.386} C_DIS
LIN {X 0.194,Y -615.990,Z 470.419,A 0.000,B 0.000,C 90.000,E1 291.354} C_DIS
LIN {X 0.142,Y -617.624,Z 470.410,A 0.000,B 0.000,C 90.000,E1 289.812} C_DIS
LIN {X -0.102,Y -619.189,Z 470.402,A 0.000,B 0.000,C 90.000,E1 288.290} C_DIS
LIN {X 0.121,Y -620.370,Z 470.394,A 0.000,B 0.000,C 90.000,E1 286.985} C_DIS
LIN {X 0.112,Y -621.832,Z 470.384,A 0.000,B 0.000,C 90.000,E1 285.190} C_DIS
LIN {X -0.213,Y -622.656,Z 470.377,A 0.000,B 0.000,C 90.000,E1 283.939} C_DIS
LIN {X 0.318,Y -623.409,Z 470.369,A 0.000,B 0.000,C 90.000,E1 282.355} C_DIS
LIN {X -0.267,Y -623.757,Z 470.362,A 0.000,B 0.000,C 90.000,E1 281.130} C_DIS
LIN {X 0.097,Y -623.972,Z 470.356,A 0.000,B 0.000,C 90.000,E1 280.074} C_DIS
LIN {X 0.030,Y -623.870,Z 470.349,A 0.000,B 0.000,C 90.000,E1 278.803} C_DIS
LIN {X -0.029,Y -623.578,Z 470.342,A 0.000,B 0.000,C 90.000,E1 277.530} C_DIS
LIN {X -0.176,Y -623.224,Z 470.338,A 0.000,B 0.000,C 90.000,E1 276.777} C_DIS
LIN {X -0.320,Y -622.443,Z 470.331,A 0.000,B 0.000,C 90.000,E1 275.511} C_DIS
LIN {X 0.145,Y -621.181,Z 470.323,A 0.000,B 0.000,C 90.000,E1 274.188} C_DIS
LIN {X -0.043,Y -619.627,Z 470.316,A 0.000,B 0.000,C 90.000,E1 272.922} C_DIS
LIN {X 0.290,Y -618.547,Z 470.312,A 0.000,B 0.000,C 90.000,E1 272.121} C_DIS
LIN {X 0.016,Y -617.323,Z 470.308,A 0.000,B 0.000,C 90.000,E1 271.375} C_DIS
LIN {X 0.013,Y -614.690,Z 470.299,A 0.000,B 0.000,C 90.000,E1 269.828} C_DIS
LIN {X -0.046,Y -611.764,Z 470.290,A 0.000,B 0.000,C 90.000,E1 268.282} C_DIS
LIN {X 0.176,Y -609.165,Z 470.283,A 0.000,B 0.000,C 90.000,E1 266.963} C_DIS
